  MoveL 3161 to (-403.79, 333.05, -22.06) mm, rotated rx -180 ry 0 rz 0.01 deg; joints [35.385, -31.602, 74.952, -134.407, 54.177, 150.081]
  MoveL 3162 to (-401.25, 328.08, -22.26) mm, rotated rx -180 ry 0 rz 0.01 deg; joints [35.301, -31.893, 75.575, -134.666, 54.367, 150.425]
  MoveL 3163 to (-395.74, 327.2, -22.47) mm, rotated rx -180 ry 0 rz 0.01 deg; joints [35.382, -32.188, 76.201, -134.749, 54.641, 150.663]
  MoveL 3164 to (-391.79, 331.15, -22.67) mm, rotated rx -180 ry 0 rz 0.01 deg; joints [35.561, -32.238, 76.316, -134.592, 54.778, 150.609]
  MoveL 3165 to (-392.66, 336.66, -22.87) mm, rotated rx 180 ry 0 rz 0.01 deg; joints [35.69, -31.995, 75.825, -134.331, 54.671, 150.312]
  MoveL 3166 to (-397.64, 339.2, -23.07) mm, rotated rx -180 ry 0 rz 0.01 deg; joints [35.663, -31.651, 75.129, -134.181, 54.411, 150.02]
  MoveL 3167 to (-398.51, 339.2, -23.1) mm, rotated rx -180 ry 0 rz 0.01 deg; joints [35.647, -31.606, 75.04, -134.175, 54.372, 149.991]
  MoveL 3168 to (-399.34, 339.13, -23.13) mm, rotated rx 180 ry 0 rz 0.01 deg; joints [35.629, -31.566, 74.959, -134.172, 54.334, 149.966]
  MoveL 3169 to (-399.69, 339.08, -23.14) mm, rotated rx 180 ry 0 rz 0.01 deg; joints [35.621, -31.55, 74.927, -134.173, 54.319, 149.957]
  MoveL 3170 to (-400.55, 338.85, -23.18) mm, rotated rx 180 ry 0 rz 0.01 deg; joints [35.599, -31.513, 74.855, -134.177, 54.282, 149.939]
  MoveL 3171 to (-400.6, 338.83, -23.18) mm, rotated rx 180 ry 0 rz 0.01 deg; joints [35.598, -31.512, 74.851, -134.178, 54.281, 149.938]
  MoveL 3172 to (-401.28, 338.49, -23.2) mm, rotated rx -180 ry 0 rz 0.01 deg; joints [35.576, -31.488, 74.805, -134.189, 54.254, 149.932]
  MoveL 3173 to (-401.4, 338.42, -23.21) mm, rotated rx -180 ry 0 rz 0.01 deg; joints [35.572, -31.484, 74.798, -134.192, 54.249, 149.932]
  MoveL 3174 to (-402.84, 337.05, -23.28) mm, rotated rx -180 ry 0 rz 0.01 deg; joints [35.509, -31.457, 74.75, -134.247, 54.202, 149.953]
  MoveL 3175 to (-402.87, 337.02, -23.28) mm, rotated rx 180 ry 0 rz 0.01 deg; joints [35.507, -31.457, 74.75, -134.249, 54.201, 149.954]
  MoveL 3176 to (-403.75, 334.43, -23.38) mm, rotated rx 180 ry 0 rz 0.01 deg; joints [35.422, -31.499, 74.848, -134.367, 54.196, 150.056]
  MoveL 3177 to (-403.78, 333.95, -23.39) mm, rotated rx 180 ry 0 rz 0.01 deg; joints [35.409, -31.514, 74.881, -134.39, 54.202, 150.08]
  MoveL 3178 to (-403.79, 333.65, -23.4) mm, rotated rx 180 ry 0 rz 0.01 deg; joints [35.401, -31.524, 74.902, -134.404, 54.206, 150.095]
  MoveL 3179 to (-403.79, 333.05, -23.43) mm, rotated rx -180 ry 0 rz 0.01 deg; joints [35.385, -31.544, 74.946, -134.434, 54.214, 150.126]
  MoveL 3180 to (-401.25, 328.08, -23.63) mm, rotated rx -180 ry 0 rz 0.01 deg; joints [35.302, -31.835, 75.57, -134.692, 54.404, 150.471]
  MoveL 3181 to (-395.74, 327.2, -23.83) mm, rotated rx -180 ry 0 rz 0.01 deg; joints [35.382, -32.13, 76.196, -134.775, 54.678, 150.709]
  MoveL 3182 to (-391.79, 331.15, -24.03) mm, rotated rx -180 ry 0 rz 0.01 deg; joints [35.562, -32.18, 76.31, -134.618, 54.815, 150.654]
  MoveL 3183 to (-392.66, 336.66, -24.23) mm, rotated rx -180 ry 0 rz 0.01 deg; joints [35.691, -31.937, 75.82, -134.357, 54.708, 150.358]
  MoveL 3184 to (-397.64, 339.2, -24.44) mm, rotated rx -180 ry 0 rz 0.01 deg; joints [35.664, -31.593, 75.124, -134.207, 54.448, 150.066]
  MoveL 3185 to (-398.51, 339.2, -24.47) mm, rotated rx -180 ry 0 rz 0.01 deg; joints [35.647, -31.549, 75.034, -134.201, 54.408, 150.036]
  MoveL 3186 to (-399.34, 339.13, -24.5) mm, rotated rx 180 ry 0 rz 0.01 deg; joints [35.63, -31.508, 74.954, -134.198, 54.371, 150.012]
  MoveL 3187 to (-399.69, 339.08, -24.51) mm, rotated rx 180 ry 0 rz 0.01 deg; joints [35.622, -31.492, 74.921, -134.199, 54.356, 150.002]
  MoveL 3188 to (-400.55, 338.85, -24.54) mm, rotated rx 180 ry 0 rz 0.01 deg; joints [35.6, -31.455, 74.849, -134.204, 54.319, 149.985]
  MoveL 3189 to (-400.6, 338.83, -24.54) mm, rotated rx 180 ry 0 rz 0.01 deg; joints [35.598, -31.454, 74.846, -134.204, 54.317, 149.984]
  MoveL 3190 to (-401.28, 338.49, -24.57) mm, rotated rx -180 ry 0 rz 0.01 deg; joints [35.577, -31.43, 74.8, -134.216, 54.29, 149.978]
  MoveL 3191 to (-401.4, 338.42, -24.57) mm, rotated rx -180 ry 0 rz 0.01 deg; joints [35.572, -31.426, 74.793, -134.218, 54.286, 149.978]
  MoveL 3192 to (-402.84, 337.05, -24.64) mm, rotated rx 180 ry 0 rz 0.01 deg; joints [35.509, -31.399, 74.744, -134.274, 54.238, 149.998]
  MoveL 3193 to (-402.87, 337.02, -24.64) mm, rotated rx -180 ry 0 rz 0.01 deg; joints [35.508, -31.399, 74.744, -134.275, 54.238, 149.999]
  MoveL 3194 to (-403.75, 334.43, -24.74) mm, rotated rx -180 ry 0 rz 0.01 deg; joints [35.423, -31.441, 74.843, -134.393, 54.233, 150.102]
  MoveL 3195 to (-403.78, 333.95, -24.76) mm, rotated rx -180 ry 0 rz 0.01 deg; joints [35.41, -31.456, 74.876, -134.417, 54.239, 150.126]
  MoveL 3196 to (-403.79, 333.65, -24.77) mm, rotated rx -180 ry 0 rz 0.01 deg; joints [35.402, -31.466, 74.896, -134.431, 54.242, 150.141]
  MoveL 3197 to (-403.79, 333.05, -24.79) mm, rotated rx -180 ry 0 rz 0.01 deg; joints [35.386, -31.486, 74.941, -134.46, 54.251, 150.172]
  MoveL 3198 to (-401.25, 328.08, -24.99) mm, rotated rx -180 ry 0 rz 0.01 deg; joints [35.302, -31.777, 75.564, -134.718, 54.441, 150.516]
  MoveL 3199 to (-395.74, 327.2, -25.19) mm, rotated rx 180 ry 0 rz 0.01 deg; joints [35.383, -32.072, 76.19, -134.8, 54.715, 150.754]
  MoveL 3200 to (-391.79, 331.15, -25.4) mm, rotated rx 180 ry 0 rz 0.01 deg; joints [35.562, -32.122, 76.305, -134.644, 54.852, 150.7]
  MoveL 3201 to (-392.66, 336.66, -25.6) mm, rotated rx -180 ry 0 rz 0.01 deg; joints [35.692, -31.879, 75.814, -134.383, 54.745, 150.403]
  MoveL 3202 to (-397.64, 339.2, -25.8) mm, rotated rx -180 ry 0 rz 0.01 deg; joints [35.664, -31.535, 75.118, -134.233, 54.485, 150.111]
  MoveL 3203 to (-398.51, 339.2, -25.83) mm, rotated rx -180 ry 0 rz 0.01 deg; joints [35.648, -31.491, 75.029, -134.227, 54.445, 150.082]
  MoveL 3204 to (-399.34, 339.13, -25.86) mm, rotated rx -180 ry 0 rz 0.01 deg; joints [35.631, -31.45, 74.948, -134.225, 54.408, 150.057]
  MoveL 3205 to (-399.69, 339.08, -25.87) mm, rotated rx 180 ry 0 rz 0.01 deg; joints [35.622, -31.434, 74.915, -134.225, 54.392, 150.048]
  MoveL 3206 to (-400.55, 338.85, -25.9) mm, rotated rx -180 ry 0 rz 0.01 deg; joints [35.6, -31.398, 74.843, -134.23, 54.356, 150.03]
  MoveL 3207 to (-400.6, 338.83, -25.91) mm, rotated rx -180 ry 0 rz 0.01 deg; joints [35.599, -31.396, 74.84, -134.23, 54.354, 150.03]
  MoveL 3208 to (-401.28, 338.49, -25.93) mm, rotated rx 180 ry 0 rz 0.01 deg; joints [35.577, -31.372, 74.794, -134.242, 54.327, 150.023]
  MoveL 3209 to (-401.4, 338.42, -25.94) mm, rotated rx -180 ry 0 rz 0.01 deg; joints [35.573, -31.369, 74.787, -134.245, 54.322, 150.023]
  MoveL 3210 to (-402.84, 337.05, -26.01) mm, rotated rx 180 ry 0 rz 0.01 deg; joints [35.51, -31.341, 74.739, -134.3, 54.275, 150.044]
  MoveL 3211 to (-402.87, 337.02, -26.01) mm, rotated rx 180 ry 0 rz 0.01 deg; joints [35.508, -31.341, 74.739, -134.301, 54.274, 150.045]
  MoveL 3212 to (-403.75, 334.43, -26.11) mm, rotated rx -180 ry 0 rz 0.01 deg; joints [35.424, -31.384, 74.837, -134.42, 54.27, 150.147]
  MoveL 3213 to (-403.78, 333.95, -26.12) mm, rotated rx 180 ry 0 rz 0.01 deg; joints [35.41, -31.398, 74.87, -134.443, 54.275, 150.171]
  MoveL 3214 to (-403.79, 333.65, -26.13) mm, rotated rx -180 ry 0 rz 0.01 deg; joints [35.403, -31.408, 74.891, -134.457, 54.279, 150.186]
  MoveL 3215 to (-403.79, 333.05, -26.15) mm, rotated rx -180 ry 0 rz 0.01 deg; joints [35.387, -31.428, 74.935, -134.486, 54.288, 150.217]
  MoveL 3216 to (-401.25, 328.08, -26.36) mm, rotated rx 180 ry 0 rz 0.01 deg; joints [35.303, -31.719, 75.558, -134.744, 54.478, 150.561]
  MoveL 3217 to (-395.74, 327.2, -26.56) mm, rotated rx -180 ry 0 rz 0.01 deg; joints [35.383, -32.013, 76.184, -134.826, 54.753, 150.799]
  MoveL 3218 to (-391.79, 331.15, -26.76) mm, rotated rx 180 ry 0 rz 0.01 deg; joints [35.563, -32.063, 76.299, -134.67, 54.89, 150.745]
  MoveL 3219 to (-392.66, 336.66, -26.96) mm, rotated rx 180 ry 0 rz 0.01 deg; joints [35.692, -31.821, 75.808, -134.409, 54.782, 150.449]
  MoveL 3220 to (-397.64, 339.2, -27.17) mm, rotated rx -180 ry 0 rz 0.01 deg; joints [35.665, -31.477, 75.112, -134.259, 54.521, 150.157]
  MoveL 3221 to (-398.51, 339.2, -27.2) mm, rotated rx -180 ry 0 rz 0.01 deg; joints [35.648, -31.433, 75.023, -134.253, 54.482, 150.127]
  MoveL 3222 to (-399.34, 339.13, -27.23) mm, rotated rx -180 ry 0 rz 0.01 deg; joints [35.631, -31.392, 74.942, -134.251, 54.444, 150.103]
  MoveL 3223 to (-399.69, 339.08, -27.24) mm, rotated rx -180 ry 0 rz 0.01 deg; joints [35.623, -31.376, 74.909, -134.251, 54.429, 150.093]
  MoveL 3224 to (-400.55, 338.85, -27.27) mm, rotated rx -180 ry 0 rz 0.01 deg; joints [35.601, -31.34, 74.837, -134.256, 54.392, 150.076]
  MoveL 3225 to (-400.6, 338.83, -27.27) mm, rotated rx -180 ry 0 rz 0.01 deg; joints [35.599, -31.338, 74.834, -134.256, 54.391, 150.075]
  MoveL 3226 to (-401.28, 338.49, -27.3) mm, rotated rx -180 ry 0 rz 0.01 deg; joints [35.578, -31.314, 74.788, -134.268, 54.364, 150.069]
  MoveL 3227 to (-401.4, 338.42, -27.3) mm, rotated rx -180 ry 0 rz 0.01 deg; joints [35.573, -31.311, 74.781, -134.271, 54.359, 150.069]
  MoveL 3228 to (-402.84, 337.05, -27.37) mm, rotated rx 180 ry 0 rz 0.01 deg; joints [35.51, -31.284, 74.733, -134.326, 54.311, 150.089]
  MoveL 3229 to (-402.87, 337.02, -27.37) mm, rotated rx -180 ry 0 rz 0.01 deg; joints [35.509, -31.283, 74.733, -134.327, 54.311, 150.09]
  MoveL 3230 to (-403.75, 334.43, -27.47) mm, rotated rx 180 ry 0 rz 0.01 deg; joints [35.424, -31.326, 74.831, -134.446, 54.306, 150.193]
  MoveL 3231 to (-403.78, 333.95, -27.49) mm, rotated rx -180 ry 0 rz 0.01 deg; joints [35.411, -31.341, 74.864, -134.469, 54.312, 150.217]
  MoveL 3232 to (-403.79, 333.65, -27.5) mm, rotated rx -180 ry 0 rz 0.01 deg; joints [35.403, -31.35, 74.885, -134.483, 54.316, 150.232]
  MoveL 3233 to (-403.79, 333.05, -27.52) mm, rotated rx 180 ry 0 rz 0.01 deg; joints [35.387, -31.37, 74.929, -134.512, 54.324, 150.263]
  MoveL 3234 to (-401.25, 328.08, -27.72) mm, rotated rx -180 ry 0 rz 0.01 deg; joints [35.303, -31.661, 75.552, -134.77, 54.515, 150.606]
  MoveL 3235 to (-395.74, 327.2, -27.92) mm, rotated rx -180 ry 0 rz 0.01 deg; joints [35.384, -31.955, 76.178, -134.852, 54.79, 150.845]
  MoveL 3236 to (-391.79, 331.15, -28.13) mm, rotated rx -180 ry 0 rz 0.01 deg; joints [35.563, -32.005, 76.293, -134.695, 54.927, 150.79]
  MoveL 3237 to (-392.66, 336.66, -28.33) mm, rotated rx 180 ry 0 rz 0.01 deg; joints [35.693, -31.763, 75.802, -134.435, 54.818, 150.494]
  MoveL 3238 to (-397.64, 339.2, -28.53) mm, rotated rx -180 ry 0 rz 0.01 deg; joints [35.665, -31.419, 75.106, -134.285, 54.558, 150.202]
  MoveL 3239 to (-398.51, 339.2, -28.56) mm, rotated rx 180 ry 0 rz 0.01 deg; joints [35.649, -31.375, 75.017, -134.279, 54.518, 150.173]
  MoveL 3240 to (-399.34, 339.13, -28.59) mm, rotated rx -180 ry 0 rz 0.01 deg; joints [35.632, -31.334, 74.936, -134.277, 54.481, 150.148]
  MoveL 3241 to (-399.69, 339.08, -28.6) mm, rotated rx 180 ry 0 rz 0.01 deg; joints [35.623, -31.318, 74.903, -134.277, 54.465, 150.139]
  MoveL 3242 to (-400.55, 338.85, -28.63) mm, rotated rx 180 ry 0 rz 0.01 deg; joints [35.601, -31.282, 74.831, -134.282, 54.429, 150.121]
  MoveL 3243 to (-400.6, 338.83, -28.64) mm, rotated rx 180 ry 0 rz 0.01 deg; joints [35.6, -31.28, 74.828, -134.282, 54.427, 150.12]
  MoveL 3244 to (-401.28, 338.49, -28.66) mm, rotated rx -180 ry 0 rz 0.01 deg; joints [35.578, -31.256, 74.782, -134.294, 54.4, 150.114]
  MoveL 3245 to (-401.4, 338.42, -28.67) mm, rotated rx -180 ry 0 rz 0.01 deg; joints [35.574, -31.253, 74.775, -134.297, 54.395, 150.114]
  MoveL 3246 to (-402.84, 337.05, -28.74) mm, rotated rx 180 ry 0 rz 0.01 deg; joints [35.511, -31.226, 74.726, -134.352, 54.348, 150.134]
  MoveL 3247 to (-402.87, 337.02, -28.74) mm, rotated rx -180 ry 0 rz 0.01 deg; joints [35.51, -31.225, 74.726, -134.353, 54.347, 150.135]
  MoveL 3248 to (-403.75, 334.43, -28.84) mm, rotated rx 180 ry 0 rz 0.01 deg; joints [35.425, -31.268, 74.825, -134.472, 54.343, 150.238]
  MoveL 3249 to (-403.78, 333.95, -28.85) mm, rotated rx 180 ry 0 rz 0.01 deg; joints [35.412, -31.282, 74.858, -134.495, 54.349, 150.262]
  MoveL 3250 to (-403.79, 333.65, -28.86) mm, rotated rx 180 ry 0 rz 0.01 deg; joints [35.404, -31.292, 74.878, -134.509, 54.352, 150.277]
  MoveL 3251 to (-403.79, 333.05, -28.88) mm, rotated rx -180 ry 0 rz 0.01 deg; joints [35.388, -31.312, 74.923, -134.538, 54.361, 150.308]
  MoveL 3252 to (-401.25, 328.08, -29.09) mm, rotated rx 180 ry 0 rz 0.01 deg; joints [35.304, -31.603, 75.546, -134.796, 54.552, 150.651]
  MoveL 3253 to (-395.74, 327.2, -29.29) mm, rotated rx 180 ry 0 rz 0.01 deg; joints [35.385, -31.897, 76.172, -134.877, 54.827, 150.89]
  MoveL 3254 to (-391.79, 331.15, -29.49) mm, rotated rx -180 ry 0 rz 0.01 deg; joints [35.564, -31.946, 76.287, -134.721, 54.964, 150.835]
  MoveL 3255 to (-392.66, 336.66, -29.69) mm, rotated rx -180 ry 0 rz 0.01 deg; joints [35.693, -31.704, 75.796, -134.46, 54.855, 150.539]
  MoveL 3256 to (-397.64, 339.2, -29.9) mm, rotated rx -180 ry 0 rz 0.01 deg; joints [35.666, -31.361, 75.1, -134.311, 54.595, 150.247]
  MoveL 3257 to (-398.51, 339.2, -29.93) mm, rotated rx 180 ry 0 rz 0.01 deg; joints [35.65, -31.316, 75.01, -134.305, 54.555, 150.218]
  MoveL 3258 to (-399.34, 339.13, -29.95) mm, rotated rx -180 ry 0 rz 0.01 deg; joints [35.632, -31.276, 74.93, -134.302, 54.517, 150.193]
  MoveL 3259 to (-399.69, 339.08, -29.97) mm, rotated rx 180 ry 0 rz 0.01 deg; joints [35.624, -31.26, 74.897, -134.303, 54.502, 150.184]
  MoveL 3260 to (-400.55, 338.85, -30) mm, rotated rx 180 ry 0 rz 0.01 deg; joints [35.602, -31.224, 74.825, -134.308, 54.465, 150.166]
  MoveL 3261 to (-400.6, 338.83, -30) mm, rotated rx 180 ry 0 rz 0.01 deg; joints [35.601, -31.222, 74.822, -134.308, 54.464, 150.166]
  MoveL 3262 to (-400.13, 339.01, -30) mm, rotated rx -180 ry 0 rz 0.01 deg; joints [35.614, -31.239, 74.856, -134.303, 54.483, 150.173]
  MoveL 3263 to (-398.92, 339.2, -30) mm, rotated rx 180 ry 0 rz 0.01 deg; joints [35.642, -31.292, 74.967, -134.303, 54.537, 150.206]
  MoveL 3264 to (-213.26, 339.2, -30) mm, rotated rx -180 ry 0 rz 0.01 deg; joints [39.465, -39.376, 91.77, -134.189, 62.458, 155.431]
  MoveL 3265 to (-213.59, 339.15, -30) mm, rotated rx -180 ry 0 rz 0.01 deg; joints [39.457, -39.365, 91.748, -134.194, 62.446, 155.425]
  MoveL 3266 to (-214.12, 339.03, -30) mm, rotated rx -180 ry 0 rz 0.01 deg; joints [39.441, -39.349, 91.713, -134.203, 62.426, 155.418]
  MoveL 3267 to (-215.21, 338.67, -30) mm, rotated rx 180 ry 0 rz 0.01 deg; joints [39.407, -39.318, 91.649, -134.225, 62.388, 155.407]
  MoveL 3268 to (-215.66, 338.49, -30) mm, rotated rx 180 ry 0 rz 0.01 deg; joints [39.392, -39.306, 91.624, -134.235, 62.373, 155.404]
  MoveL 3269 to (-226.55, 333.14, -30) mm, rotated rx 180 ry 0 rz 0.01 deg; joints [39.004, -39.05, 91.096, -134.527, 62.012, 155.373]
  MoveL 3270 to (-227.09, 332.81, -30) mm, rotated rx -180 ry 0 rz 0.01 deg; joints [38.983, -39.039, 91.074, -134.545, 61.995, 155.374]
  MoveL 3271 to (-228.18, 331.99, -30) mm, rotated rx 180 ry 0 rz 0.01 deg; joints [38.936, -39.022, 91.039, -134.585, 61.962, 155.382]
  MoveL 3272 to (-228.47, 331.74, -30) mm, rotated rx 180 ry 0 rz 0.01 deg; joints [38.923, -39.018, 91.032, -134.597, 61.954, 155.386]
  MoveL 3273 to (-236.6, 324.01, -30) mm, rotated rx -180 ry 0 rz 0.01 deg; joints [38.532, -38.937, 90.874, -134.967, 61.729, 155.516]
  MoveL 3274 to (-236.83, 323.76, -30) mm, rotated rx 180 ry 0 rz 0.01 deg; joints [38.52, -38.936, 90.871, -134.978, 61.722, 155.521]
  MoveL 3275 to (-237.77, 322.67, -30) mm, rotated rx 180 ry 0 rz 0.01 deg; joints [38.47, -38.932, 90.865, -135.029, 61.699, 155.544]
  MoveL 3276 to (-238.12, 322.17, -30) mm, rotated rx -180 ry 0 rz 0.01 deg; joints [38.449, -38.934, 90.868, -135.052, 61.691, 155.556]
  MoveL 3277 to (-240.45, 318.18, -30) mm, rotated rx -180 ry 0 rz 0.01 deg; joints [38.288, -38.963, 90.937, -135.231, 61.649, 155.667]
  MoveL 3278 to (-240.5, 318.08, -30) mm, rotated rx -180 ry 0 rz 0.01 deg; joints [38.284, -38.964, 90.938, -135.235, 61.648, 155.67]
  MoveL 3279 to (-244.03, 311.56, -30) mm, rotated rx -180 ry 0 rz 0.01 deg; joints [38.027, -39.023, 91.07, -135.526, 61.589, 155.856]
  MoveL 3280 to (-244.21, 311.15, -30) mm, rotated rx -180 ry 0 rz 0.01 deg; joints [38.012, -39.027, 91.081, -135.544, 61.586, 155.868]
  MoveL 3281 to (-244.76, 309.7, -30) mm, rotated rx 180 ry 0 rz 0.01 deg; joints [37.96, -39.049, 91.129, -135.607, 61.582, 155.915]
  MoveL 3282 to (-244.95, 309.01, -30) mm, rotated rx 180 ry 0 rz 0.01 deg; joints [37.936, -39.063, 91.158, -135.637, 61.584, 155.939]
  MoveL 3283 to (-246.39, 299.58, -30) mm, rotated rx -180 ry 0 rz 0.01 deg; joints [37.643, -39.287, 91.642, -136.037, 61.644, 156.292]
  MoveL 3284 to (-246.42, 299.36, -30) mm, rotated rx -180 ry 0 rz 0.01 deg; joints [37.636, -39.293, 91.654, -136.046, 61.646, 156.3]
  MoveL 3285 to (-246.51, 298.27, -30) mm, rotated rx 180 ry 0 rz 0.01 deg; joints [37.603, -39.321, 91.715, -136.092, 61.656, 156.342]
  MoveC 3286 to (-246.51, 297.75, -30) mm, rotated rx -180 ry 0 rz 0.01 deg; joints [37.589, -39.336, 91.748, -136.113, 61.662, 156.363] to (-246.44, 297.24, -30) mm, rotated rx 180 ry 0 rz 0.01 deg; joints [37.576, -39.354, 91.786, -136.134, 61.672, 156.385]
  MoveL 3287 to (-245.04, 290.99, -30) mm, rotated rx 180 ry 0 rz 0.01 deg; joints [37.431, -39.593, 92.296, -136.384, 61.806, 156.671]
  MoveL 3288 to (-245.03, 290.92, -30) mm, rotated rx -180 ry 0 rz 0.01 deg; joints [37.429, -39.596, 92.301, -136.387, 61.808, 156.674]
  MoveL 3289 to (-244.07, 287.01, -30) mm, rotated rx 180 ry 0 rz 0.01 deg; joints [37.34, -39.747, 92.625, -136.543, 61.895, 156.852]
  MoveL 3290 to (-243.75, 286.2, -30) mm, rotated rx 180 ry 0 rz 0.01 deg; joints [37.324, -39.783, 92.702, -136.574, 61.918, 156.892]
  MoveL 3291 to (-241.96, 282.93, -30) mm, rotated rx -180 ry 0 rz 0.01 deg; joints [37.27, -39.948, 93.051, -136.698, 62.031, 157.063]
  MoveL 3292 to (-241.77, 282.61, -30) mm, rotated rx -180 ry 0 rz 0.01 deg; joints [37.265, -39.965, 93.088, -136.71, 62.043, 157.08]
  MoveL 3293 to (-239.73, 279.71, -30) mm, rotated rx -180 ry 0 rz 0.01 deg; joints [37.227, -40.128, 93.434, -136.816, 62.16, 157.241]
  MoveL 3294 to (-239.54, 279.46, -30) mm, rotated rx -180 ry 0 rz 0.01 deg; joints [37.224, -40.142, 93.464, -136.824, 62.171, 157.255]
  MoveL 3295 to (-237.07, 276.56, -30) mm, rotated rx -180 ry 0 rz 0.01 deg; joints [37.194, -40.321, 93.844, -136.927, 62.306, 157.425]
  MoveL 3296 to (-236.53, 276.05, -30) mm, rotated rx -180 ry 0 rz 0.01 deg; joints [37.192, -40.356, 93.919, -136.944, 62.333, 157.457]
  MoveL 3297 to (-232.69, 273.15, -30) mm, rotated rx -180 ry 0 rz 0.01 deg; joints [37.192, -40.587, 94.408, -137.036, 62.523, 157.655]
  MoveL 3298 to (-232.49, 273.01, -30) mm, rotated rx 180 ry 0 rz 0.01 deg; joints [37.192, -40.599, 94.433, -137.04, 62.532, 157.665]
  MoveL 3299 to (-229.8, 271.26, -30) mm, rotated rx 180 ry 0 rz 0.01 deg; joints [37.201, -40.752, 94.757, -137.092, 62.661, 157.792]
  MoveL 3300 to (-229.47, 271.08, -30) mm, rotated rx 180 ry 0 rz 0.01 deg; joints [37.203, -40.769, 94.794, -137.097, 62.676, 157.806]
  MoveL 3301 to (-227.17, 269.92, -30) mm, rotated rx -180 ry 0 rz 0.01 deg; joints [37.22, -40.89, 95.049, -137.126, 62.782, 157.901]
  MoveL 3302 to (-226.75, 269.75, -30) mm, rotated rx -180 ry 0 rz 0.01 deg; joints [37.224, -40.911, 95.093, -137.13, 62.8, 157.917]
  MoveL 3303 to (-223.98, 268.79, -30) mm, rotated rx 180 ry 0 rz 0.01 deg; joints [37.257, -41.043, 95.374, -137.148, 62.921, 158.014]
  MoveL 3304 to (-223.48, 268.66, -30) mm, rotated rx -180 ry 0 rz 0.01 deg; joints [37.264, -41.066, 95.421, -137.149, 62.943, 158.03]
  MoveL 3305 to (-219.13, 267.87, -30) mm, rotated rx 180 ry 0 rz 0.01 deg; joints [37.337, -41.253, 95.816, -137.146, 63.124, 158.154]
  MoveL 3306 to (-218.95, 267.85, -30) mm, rotated rx 180 ry 0 rz 0.01 deg; joints [37.34, -41.261, 95.832, -137.146, 63.131, 158.159]
  MoveL 3307 to (-215.32, 267.39, -30) mm, rotated rx 180 ry 0 rz 0.01 deg; joints [37.406, -41.41, 96.148, -137.134, 63.279, 158.253]
  MoveL 3308 to (-214.9, 267.36, -30) mm, rotated rx 180 ry 0 rz 0.01 deg; joints [37.415, -41.427, 96.183, -137.131, 63.296, 158.263]
  MoveL 3309 to (-178.62, 267.36, -30) mm, rotated rx -180 ry 0 rz 0.01 deg; joints [38.23, -42.764, 99.002, -136.789, 64.694, 159.014]
  MoveL 3310 to (-178.19, 267.39, -30) mm, rotated rx 180 ry 0 rz 0.01 deg; joints [38.24, -42.778, 99.033, -136.784, 64.71, 159.021]
  MoveL 3311 to (-174.57, 267.85, -30) mm, rotated rx -180 ry 0 rz 0.01 deg; joints [38.336, -42.896, 99.282, -136.727, 64.842, 159.077]
  MoveL 3312 to (-174.39, 267.87, -30) mm, rotated rx 180 ry 0 rz 0.01 deg; joints [38.341, -42.902, 99.294, -136.724, 64.849, 159.08]
  MoveL 3313 to (-170.03, 268.66, -30) mm, rotated rx -180 ry 0 rz 0.01 deg; joints [38.465, -43.036, 99.577, -136.646, 65.003, 159.138]
  MoveL 3314 to (-169.59, 268.78, -30) mm, rotated rx 180 ry 0 rz 0.01 deg; joints [38.478, -43.049, 99.604, -136.637, 65.019, 159.142]
  MoveL 3315 to (-167.47, 269.46, -30) mm, rotated rx -180 ry 0 rz 0.01 deg; joints [38.547, -43.106, 99.722, -136.586, 65.09, 159.159]
  MoveL 3316 to (-167.12, 269.6, -30) mm, rotated rx 180 ry 0 rz 0.01 deg; joints [38.559, -43.115, 99.74, -136.577, 65.101, 159.161]
  MoveL 3317 to (-164.88, 270.63, -30) mm, rotated rx 180 ry 0 rz 0.01 deg; joints [38.641, -43.166, 99.848, -136.511, 65.173, 159.167]
  MoveL 3318 to (-164.5, 270.83, -30) mm, rotated rx -180 ry 0 rz 0.01 deg; joints [38.656, -43.174, 99.864, -136.499, 65.184, 159.167]
  MoveL 3319 to (-161.59, 272.64, -30) mm, rotated rx 180 ry 0 rz 0.01 deg; joints [38.776, -43.227, 99.974, -136.395, 65.271, 159.158]
  MoveL 3320 to (-161.36, 272.79, -30) mm, rotated rx 180 ry 0 rz 0.01 deg; joints [38.786, -43.231, 99.982, -136.386, 65.277, 159.156]
  MoveL 3321 to (-157, 276.04, -30) mm, rotated rx 180 ry 0 rz 0.01 deg; joints [38.981, -43.295, 100.113, -136.208, 65.4, 159.122]
  MoveL 3322 to (-156.45, 276.55, -30) mm, rotated rx 180 ry 0 rz 0.01 deg; joints [39.009, -43.301, 100.123, -136.181, 65.414, 159.113]
  MoveL 3323 to (-154.49, 278.84, -30) mm, rotated rx 180 ry 0 rz 0.01 deg; joints [39.121, -43.306, 100.131, -136.067, 65.458, 159.066]
  MoveL 3324 to (-154.32, 279.05, -30) mm, rotated rx 180 ry 0 rz 0.01 deg; joints [39.131, -43.306, 100.13, -136.057, 65.462, 159.062]
  MoveL 3325 to (-151.94, 282.32, -30) mm, rotated rx -180 ry 0 rz 0.01 deg; joints [39.282, -43.298, 100.109, -135.9, 65.509, 158.987]
  MoveL 3326 to (-151.71, 282.67, -30) mm, rotated rx 180 ry 0 rz 0.01 deg; joints [39.297, -43.296, 100.105, -135.884, 65.513, 158.978]
  MoveL 3327 to (-149.77, 286.18, -30) mm, rotated rx 180 ry 0 rz 0.01 deg; joints [39.444, -43.266, 100.035, -135.722, 65.541, 158.885]
  MoveL 3328 to (-149.44, 287.04, -30) mm, rotated rx -180 ry 0 rz 0.01 deg; joints [39.477, -43.254, 100.008, -135.684, 65.543, 158.859]
  MoveL 3329 to (-147.12, 296.83, -30) mm, rotated rx 180 ry 0 rz 0.01 deg; joints [39.812, -43.058, 99.578, -135.27, 65.505, 158.534]
  MoveL 3330 to (-147.03, 297.45, -30) mm, rotated rx -180 ry 0 rz 0.01 deg; joints [39.831, -43.043, 99.546, -135.244, 65.501, 158.513]
  MoveL 3331 to (-146.99, 298.18, -30) mm, rotated rx 180 ry 0 rz 0.01 deg; joints [39.853, -43.024, 99.504, -135.215, 65.493, 158.486]
  MoveL 3332 to (-147.03, 298.84, -30) mm, rotated rx 180 ry 0 rz 0.01 deg; joints [39.871, -43.004, 99.46, -135.19, 65.483, 158.46]
  MoveL 3333 to (-148.48, 308.63, -30) mm, rotated rx -180 ry 0 rz 0.01 deg; joints [40.114, -42.671, 98.742, -134.819, 65.306, 158.055]
  MoveL 3334 to (-148.63, 309.25, -30) mm, rotated rx -180 ry 0 rz 0.01 deg; joints [40.128, -42.647, 98.692, -134.796, 65.293, 158.028]
  MoveL 3335 to (-149.27, 311.07, -30) mm, rotated rx -180 ry 0 rz 0.01 deg; joints [40.164, -42.572, 98.53, -134.732, 65.246, 157.945]
  MoveL 3336 to (-149.48, 311.55, -30) mm, rotated rx -180 ry 0 rz 0.01 deg; joints [40.172, -42.551, 98.484, -134.715, 65.232, 157.922]
  MoveL 3337 to (-151.43, 315.17, -30) mm, rotated rx 180 ry 0 rz 0.01 deg; joints [40.228, -42.376, 98.11, -134.593, 65.115, 157.742]
  MoveL 3338 to (-151.46, 315.23, -30) mm, rotated rx -180 ry 0 rz 0.01 deg; joints [40.229, -42.373, 98.105, -134.591, 65.113, 157.739]
  MoveL 3339 to (-155.12, 321.76, -30) mm, rotated rx 180 ry 0 rz 0.01 deg; joints [40.325, -42.051, 97.416, -134.373, 64.894, 157.408]
  MoveL 3340 to (-155.44, 322.24, -30) mm, rotated rx 180 ry 0 rz 0.01 deg; joints [40.33, -42.026, 97.361, -134.357, 64.876, 157.383]
  MoveL 3341 to (-156.62, 323.69, -30) mm, rotated rx -180 ry 0 rz 0.01 deg; joints [40.343, -41.941, 97.18, -134.312, 64.814, 157.301]
  MoveL 3342 to (-156.92, 324.01, -30) mm, rotated rx -180 ry 0 rz 0.01 deg; joints [40.345, -41.921, 97.138, -134.303, 64.799, 157.283]
  MoveL 3343 to (-165.04, 331.74, -30) mm, rotated rx -180 ry 0 rz 0.01 deg; joints [40.368, -41.398, 96.026, -134.079, 64.398, 156.805]
  MoveL 3344 to (-165.34, 331.99, -30) mm, rotated rx -180 ry 0 rz 0.01 deg; joints [40.368, -41.38, 95.987, -134.072, 64.384, 156.789]
  MoveL 3345 to (-166.42, 332.81, -30) mm, rotated rx 180 ry 0 rz 0.01 deg; joints [40.365, -41.316, 95.851, -134.05, 64.333, 156.733]
  MoveL 3346 to (-166.97, 333.14, -30) mm, rotated rx -180 ry 0 rz 0.01 deg; joints [40.361, -41.286, 95.789, -134.042, 64.308, 156.708]
  MoveL 3347 to (-177.85, 338.49, -30) mm, rotated rx -180 ry 0 rz 0.01 deg; joints [40.254, -40.727, 94.606, -133.931, 63.83, 156.257]
  MoveL 3348 to (-178.19, 338.64, -30) mm, rotated rx 180 ry 0 rz 0.01 deg; joints [40.251, -40.711, 94.57, -133.929, 63.815, 156.244]
  MoveL 3349 to (-178.91, 338.9, -30) mm, rotated rx -180 ry 0 rz 0.01 deg; joints [40.241, -40.676, 94.497, -133.925, 63.784, 156.217]
  MoveL 3350 to (-179.55, 339.06, -30) mm, rotated rx 180 ry 0 rz 0.01 deg; joints [40.231, -40.648, 94.437, -133.924, 63.758, 156.196]
  MoveL 3351 to (-180.46, 339.2, -30) mm, rotated rx 180 ry 0 rz 0.01 deg; joints [40.213, -40.61, 94.357, -133.927, 63.722, 156.171]
  MoveL 3352 to (4.87, 339.21, -30) mm, rotated rx -180 ry 0 rz 0.01 deg; joints [44.913, -46.774, 107.418, -131.39, 70.267, 159.8]
  MoveL 3353 to (5.94, 339.15, -30) mm, rotated rx 180 ry 0 rz 0.01 deg; joints [44.941, -46.808, 107.491, -131.373, 70.303, 159.821]
  MoveL 3354 to (6.8, 338.95, -30) mm, rotated rx 180 ry 0 rz 0.01 deg; joints [44.959, -46.84, 107.559, -131.364, 70.333, 159.843]
  MoveL 3355 to (7.07, 338.84, -30) mm, rotated rx -180 ry 0 rz 0.01 deg; joints [44.963, -46.851, 107.583, -131.363, 70.344, 159.852]
  MoveL 3356 to (7.37, 338.63, -30) mm, rotated rx -180 ry 0 rz 0.01 deg; joints [44.966, -46.866, 107.616, -131.365, 70.356, 159.865]
  MoveL 3357 to (9.66, 336.38, -30) mm, rotated rx 180 ry 0 rz 0.01 deg; joints [44.967, -47, 107.906, -131.406, 70.46, 159.99]
  MoveL 3358 to (9.9, 336.02, -30) mm, rotated rx 180 ry 0 rz 0.01 deg; joints [44.963, -47.018, 107.944, -131.415, 70.472, 160.007]
  MoveL 3359 to (10.07, 335.56, -30) mm, rotated rx 180 ry 0 rz 0.01 deg; joints [44.955, -47.036, 107.984, -131.429, 70.484, 160.027]
  MoveL 3360 to (10.27, 334.35, -30) mm, rotated rx 180 ry 0 rz 0.01 deg; joints [44.927, -47.077, 108.074, -131.47, 70.506, 160.075]
  MoveL 3361 to (10.27, 31.84, -30) mm, rotated rx -180 ry 0 rz 0.01 deg; joints [35.126, -54.404, 124.671, -143.341, 74.579, 169.75]
  MoveL 3362 to (9.14, 36.48, -30) mm, rotated rx 180 ry 0 rz 0.01 deg; joints [35.269, -54.28, 124.38, -143.169, 74.475, 169.606]
  MoveL 3363 to (9.02, 36.86, -30) mm, rotated rx -180 ry 0 rz 0.01 deg; joints [35.28, -54.268, 124.354, -143.155, 74.466, 169.594]
  MoveL 3364 to (8.51, 38.24, -30) mm, rotated rx -180 ry 0 rz 0.01 deg; joints [35.317, -54.226, 124.256, -143.107, 74.428, 169.549]
  MoveL 3365 to (8.27, 38.74, -30) mm, rotated rx 180 ry 0 rz 0.01 deg; joints [35.33, -54.209, 124.217, -143.091, 74.413, 169.531]
  MoveL 3366 to (6.11, 42.48, -30) mm, rotated rx 180 ry 0 rz 0.01 deg; joints [35.411, -54.071, 123.899, -142.978, 74.286, 169.396]
  MoveL 3367 to (6.06, 42.56, -30) mm, rotated rx -180 ry 0 rz 0.01 deg; joints [35.413, -54.068, 123.892, -142.976, 74.283, 169.393]
  MoveL 3368 to (2.27, 48.73, -30) mm, rotated rx -180 ry 0 rz 0.01 deg; joints [35.54, -53.832, 123.35, -142.794, 74.066, 169.164]
  MoveL 3369 to (2.07, 49.02, -30) mm, rotated rx -180 ry 0 rz 0.01 deg; joints [35.545, -53.82, 123.323, -142.786, 74.055, 169.153]
  MoveL 3370 to (1.04, 50.35, -30) mm, rotated rx 180 ry 0 rz 0.01 deg; joints [35.567, -53.763, 123.192, -142.751, 74.001, 169.1]
  MoveL 3371 to (0.49, 50.92, -30) mm, rotated rx 180 ry 0 rz 0.01 deg; joints [35.573, -53.735, 123.128, -142.738, 73.974, 169.076]
  MoveL 3372 to (-7.44, 57.29, -30) mm, rotated rx -180 ry 0 rz 0.01 deg; joints [35.599, -53.37, 122.299, -142.631, 73.61, 168.775]
  MoveL 3373 to (-7.81, 57.56, -30) mm, rotated rx 180 ry 0 rz 0.01 deg; joints [35.599, -53.353, 122.261, -142.627, 73.593, 168.762]
  MoveL 3374 to (-8.48, 57.96, -30) mm, rotated rx -180 ry 0 rz 0.01 deg; joints [35.596, -53.325, 122.198, -142.624, 73.565, 168.74]
  MoveL 3375 to (-9.25, 58.3, -30) mm, rotated rx 180 ry 0 rz 0.01 deg; joints [35.589, -53.295, 122.13, -142.625, 73.533, 168.719]
  MoveL 3376 to (-19.1, 61.27, -30) mm, rotated rx -180 ry 0 rz 0.01 deg; joints [35.442, -52.937, 121.329, -142.693, 73.148, 168.482]
  MoveL 3377 to (-20, 61.42, -30) mm, rotated rx 180 ry 0 rz 0.01 deg; joints [35.425, -52.907, 121.262, -142.704, 73.115, 168.464]
  MoveL 3378 to (-23.26, 61.5, -30) mm, rotated rx 180 ry 0 rz 0.01 deg; joints [35.344, -52.807, 121.038, -142.763, 72.999, 168.411]
  MoveL 3379 to (-23.6, 61.49, -30) mm, rotated rx 180 ry 0 rz 0.01 deg; joints [35.335, -52.797, 121.016, -142.77, 72.987, 168.406]
  MoveL 3380 to (-27.23, 61.21, -30) mm, rotated rx 180 ry 0 rz 0.01 deg; joints [35.233, -52.692, 120.784, -142.851, 72.863, 168.358]
  MoveL 3381 to (-27.55, 61.17, -30) mm, rotated rx 180 ry 0 rz 0.01 deg; joints [35.224, -52.683, 120.765, -142.859, 72.853, 168.354]
  MoveL 3382 to (-31.54, 60.47, -30) mm, rotated rx 180 ry 0 rz 0.01 deg; joints [35.098, -52.575, 120.528, -142.962, 72.721, 168.312]
  MoveL 3383 to (-32.27, 60.26, -30) mm, rotated rx -180 ry 0 rz 0.01 deg; joints [35.072, -52.557, 120.488, -142.985, 72.698, 168.306]
  MoveL 3384 to (-36.67, 58.42, -30) mm, rotated rx 180 ry 0 rz 0.01 deg; joints [34.896, -52.46, 120.277, -143.143, 72.567, 168.29]
  MoveL 3385 to (-36.89, 58.31, -30) mm, rotated rx 180 ry 0 rz 0.01 deg; joints [34.886, -52.455, 120.267, -143.152, 72.561, 168.29]
  MoveL 3386 to (-40.11, 56.68, -30) mm, rotated rx 180 ry 0 rz 0.01 deg; joints [34.748, -52.389, 120.125, -143.279, 72.468, 168.286]
  MoveL 3387 to (-40.47, 56.47, -30) mm, rotated rx -180 ry 0 rz 0.01 deg; joints [34.731, -52.383, 120.11, -143.295, 72.458, 168.286]
  MoveL 3388 to (-42.35, 55.2, -30) mm, rotated rx -180 ry 0 rz 0.01 deg; joints [34.639, -52.35, 120.042, -143.382, 72.408, 168.293]
  MoveL 3389 to (-42.66, 54.97, -30) mm, rotated rx 180 ry 0 rz 0.01 deg; joints [34.623, -52.346, 120.032, -143.397, 72.4, 168.295]
  MoveL 3390 to (-44.72, 53.2, -30) mm, rotated rx 180 ry 0 rz 0.01 deg; joints [34.509, -52.318, 119.974, -143.508, 72.351, 168.313]
  MoveL 3391 to (-45.04, 52.88, -30) mm, rotated rx 180 ry 0 rz 0.01 deg; joints [34.489, -52.314, 119.967, -143.527, 72.343, 168.317]
  MoveL 3392 to (-46.91, 50.78, -30) mm, rotated rx -180 ry 0 rz 0.01 deg; joints [34.368, -52.299, 119.937, -143.649, 72.304, 168.347]
  MoveL 3393 to (-47.05, 50.61, -30) mm, rotated rx -180 ry 0 rz 0.01 deg; joints [34.358, -52.298, 119.935, -143.659, 72.302, 168.349]
  MoveL 3394 to (-50.38, 46.34, -30) mm, rotated rx 180 ry 0 rz 0.01 deg; joints [34.123, -52.28, 119.906, -143.897, 72.239, 168.418]
  MoveL 3395 to (-50.64, 45.95, -30) mm, rotated rx -180 ry 0 rz 0.01 deg; joints [34.103, -52.28, 119.906, -143.918, 72.235, 168.425]
  MoveL 3396 to (-68.79, 14.55, -30) mm, rotated rx 180 ry 0 rz 0.01 deg; joints [32.525, -52.325, 120.077, -145.558, 71.991, 169.014]
  MoveL 3397 to (-68.98, 14.18, -30) mm, rotated rx 180 ry 0 rz 0.01 deg; joints [32.507, -52.327, 120.08, -145.577, 71.989, 169.022]
  MoveL 3398 to (-70.67, 10.19, -30) mm, rotated rx -180 ry 0 rz 0.01 deg; joints [32.321, -52.349, 120.139, -145.775, 71.98, 169.104]
  MoveL 3399 to (-70.75, 9.99, -30) mm, rotated rx -180 ry 0 rz 0.01 deg; joints [32.312, -52.35, 120.142, -145.785, 71.979, 169.109]
  MoveL 3400 to (-72.02, 6.36, -30) mm, rotated rx 180 ry 0 rz 0.01 deg; joints [32.148, -52.379, 120.213, -145.961, 71.98, 169.187]
  MoveL 3401 to (-72.14, 5.94, -30) mm, rotated rx -180 ry 0 rz 0.01 deg; joints [32.13, -52.383, 120.223, -145.981, 71.981, 169.197]
  MoveL 3402 to (-72.6, 3.77, -30) mm, rotated rx 180 ry 0 rz 0.01 deg; joints [32.039, -52.409, 120.286, -146.081, 71.992, 169.249]
  MoveL 3403 to (-72.66, 3.38, -30) mm, rotated rx 180 ry 0 rz 0.01 deg; joints [32.023, -52.415, 120.299, -146.099, 71.995, 169.258]
  MoveL 3404 to (-72.93, 0.48, -30) mm, rotated rx -180 ry 0 rz 0.01 deg; joints [31.909, -52.46, 120.408, -146.227, 72.023, 169.332]
  MoveL 3405 to (-72.94, 0.01, -30) mm, rotated rx 180 ry 0 rz 0.01 deg; joints [31.891, -52.469, 120.427, -146.247, 72.029, 169.345]
  MoveL 3406 to (-72.81, -2.9, -30) mm, rotated rx -180 ry 0 rz 0.01 deg; joints [31.787, -52.527, 120.563, -146.369, 72.072, 169.424]
  MoveL 3407 to (-72.79, -3.12, -30) mm, rotated rx -180 ry 0 rz 0.01 deg; joints [31.779, -52.532, 120.574, -146.378, 72.075, 169.43]
  MoveL 3408 to (-72.17, -8.56, -30) mm, rotated rx 180 ry 0 rz 0.01 deg; joints [31.59, -52.652, 120.854, -146.601, 72.169, 169.584]
  MoveL 3409 to (-72, -9.3, -30) mm, rotated rx 180 ry 0 rz 0.01 deg; joints [31.566, -52.671, 120.898, -146.63, 72.185, 169.607]
  MoveL 3410 to (-70.79, -12.74, -30) mm, rotated rx 180 ry 0 rz 0.01 deg; joints [31.465, -52.773, 121.131, -146.757, 72.275, 169.715]
  MoveL 3411 to (-70.68, -13.03, -30) mm, rotated rx -180 ry 0 rz 0.01 deg; joints [31.457, -52.782, 121.152, -146.767, 72.283, 169.725]
  MoveL 3412 to (-69.26, -16.12, -30) mm, rotated rx 180 ry 0 rz 0.01 deg; joints [31.373, -52.883, 121.384, -146.876, 72.376, 169.827]
  MoveL 3413 to (-69.12, -16.4, -30) mm, rotated rx 180 ry 0 rz 0.01 deg; joints [31.366, -52.893, 121.406, -146.886, 72.385, 169.836]
  MoveL 3414 to (-67.66, -18.94, -30) mm, rotated rx 180 ry 0 rz 0.01 deg; joints [31.304, -52.985, 121.617, -146.97, 72.472, 169.924]
  MoveL 3415 to (-67.52, -19.15, -30) mm, rotated rx 180 ry 0 rz 0.01 deg; joints [31.299, -52.993, 121.636, -146.977, 72.48, 169.932]
  MoveL 3416 to (-66.77, -20.26, -30) mm, rotated rx -180 ry 0 rz 0.01 deg; joints [31.274, -53.037, 121.736, -147.012, 72.522, 169.972]
  MoveL 3417 to (-66.29, -20.83, -30) mm, rotated rx -180 ry 0 rz 0.01 deg; joints [31.264, -53.062, 121.794, -147.028, 72.547, 169.994]
  MoveL 3418 to (-59.76, -26.97, -30) mm, rotated rx 180 ry 0 rz 0.01 deg; joints [31.18, -53.378, 122.512, -147.182, 72.869, 170.249]
  MoveL 3419 to (-59.61, -27.11, -30) mm, rotated rx 180 ry 0 rz 0.01 deg; joints [31.179, -53.385, 122.529, -147.185, 72.877, 170.255]
  MoveL 3420 to (-58.52, -28.02, -30) mm, rotated rx 180 ry 0 rz 0.01 deg; joints [31.169, -53.436, 122.644, -147.206, 72.929, 170.295]
  MoveC 3421 to (-58.08, -28.32, -30) mm, rotated rx 180 ry 0 rz 0.01 deg; joints [31.168, -53.455, 122.687, -147.211, 72.949, 170.309] to (-57.61, -28.56, -30) mm, rotated rx -180 ry 0 rz 0.01 deg; joints [31.17, -53.474, 122.73, -147.213, 72.97, 170.322]
  MoveL 3422 to (-50.81, -31.27, -30) mm, rotated rx 180 ry 0 rz 0.01 deg; joints [31.224, -53.734, 123.319, -147.212, 73.256, 170.491]
  MoveL 3423 to (-342.73, -31.27, -30) mm, rotated rx -180 ry 0 rz 0.01 deg; joints [25.555, -43.349, 100.769, -150.599, 61.537, 166.051]
  MoveL 3424 to (-336.29, -28.75, -30) mm, rotated rx 180 ry 0 rz 0.01 deg; joints [25.744, -43.563, 101.219, -150.454, 61.792, 166.082]
  MoveL 3425 to (-335.78, -28.51, -30) mm, rotated rx 180 ry 0 rz 0.01 deg; joints [25.761, -43.579, 101.253, -150.44, 61.812, 166.083]
  MoveL 3426 to (-335.06, -28.07, -30) mm, rotated rx 180 ry 0 rz 0.01 deg; joints [25.787, -43.6, 101.297, -150.417, 61.839, 166.082]
  MoveL 3427 to (-334.48, -27.64, -30) mm, rotated rx 180 ry 0 rz 0.01 deg; joints [25.811, -43.615, 101.328, -150.395, 61.859, 166.079]
  MoveL 3428 to (-327.59, -21.19, -30) mm, rotated rx 180 ry 0 rz 0.01 deg; joints [26.142, -43.772, 101.649, -150.077, 62.089, 165.997]
  MoveL 3429 to (-327.4, -20.99, -30) mm, rotated rx 180 ry 0 rz 0.01 deg; joints [26.152, -43.776, 101.657, -150.067, 62.095, 165.995]
  MoveL 3430 to (-326.75, -20.28, -30) mm, rotated rx -180 ry 0 rz 0.01 deg; joints [26.187, -43.789, 101.683, -150.032, 62.116, 165.984]
  MoveL 3431 to (-326.35, -19.74, -30) mm, rotated rx 180 ry 0 rz 0.01 deg; joints [26.212, -43.795, 101.694, -150.007, 62.127, 165.974]
  MoveL 3432 to (-324.6, -16.81, -30) mm, rotated rx 180 ry 0 rz 0.01 deg; joints [26.34, -43.81, 101.72, -149.87, 62.171, 165.913]
  MoveL 3433 to (-324.44, -16.49, -30) mm, rotated rx 180 ry 0 rz 0.01 deg; joints [26.354, -43.81, 101.721, -149.856, 62.175, 165.907]
  MoveL 3434 to (-322.84, -13.04, -30) mm, rotated rx 180 ry 0 rz 0.01 deg; joints [26.497, -43.809, 101.711, -149.697, 62.206, 165.828]
  MoveL 3435 to (-322.72, -12.74, -30) mm, rotated rx 180 ry 0 rz 0.01 deg; joints [26.509, -43.808, 101.709, -149.684, 62.208, 165.82]
  MoveL 3436 to (-321.51, -9.3, -30) mm, rotated rx 180 ry 0 rz 0.01 deg; joints [26.645, -43.791, 101.666, -149.529, 62.222, 165.735]
  MoveL 3437 to (-321.34, -8.56, -30) mm, rotated rx 180 ry 0 rz 0.01 deg; joints [26.673, -43.784, 101.649, -149.496, 62.221, 165.715]
  MoveL 3438 to (-320.72, -3.12, -30) mm, rotated rx 180 ry 0 rz 0.01 deg; joints [26.866, -43.704, 101.469, -149.259, 62.187, 165.557]
  MoveL 3439 to (-320.7, -2.9, -30) mm, rotated rx -180 ry 0 rz 0.01 deg; joints [26.874, -43.7, 101.46, -149.249, 62.185, 165.551]
  MoveL 3440 to (-320.57, 0.01, -30) mm, rotated rx 180 ry 0 rz 0.01 deg; joints [26.973, -43.649, 101.347, -149.124, 62.159, 165.463]
  MoveL 3441 to (-320.58, 0.42, -30) mm, rotated rx 180 ry 0 rz 0.01 deg; joints [26.987, -43.641, 101.329, -149.107, 62.154, 165.45]
  MoveL 3442 to (-320.74, 2.59, -30) mm, rotated rx -180 ry 0 rz 0.01 deg; joints [27.057, -43.592, 101.221, -149.014, 62.122, 165.379]
  MoveL 3443 to (-320.79, 2.99, -30) mm, rotated rx 180 ry 0 rz 0.01 deg; joints [27.069, -43.582, 101.199, -148.998, 62.116, 165.366]
  MoveL 3444 to (-321.36, 5.89, -30) mm, rotated rx 180 ry 0 rz 0.01 deg; joints [27.156, -43.503, 101.025, -148.877, 62.059, 165.265]
  MoveL 3445 to (-321.49, 6.36, -30) mm, rotated rx -180 ry 0 rz 0.01 deg; joints [27.169, -43.489, 100.994, -148.858, 62.048, 165.248]
  MoveL 3446 to (-322.72, 9.87, -30) mm, rotated rx -180 ry 0 rz 0.01 deg; joints [27.265, -43.371, 100.737, -148.715, 61.955, 165.117]
  MoveL 3447 to (-322.79, 10.06, -30) mm, rotated rx 180 ry 0 rz 0.01 deg; joints [27.27, -43.364, 100.722, -148.708, 61.95, 165.109]
  MoveL 3448 to (-324.35, 13.8, -30) mm, rotated rx 180 ry 0 rz 0.01 deg; joints [27.368, -43.227, 100.425, -148.557, 61.84, 164.964]
  MoveL 3449 to (-324.54, 14.18, -30) mm, rotated rx -180 ry 0 rz 0.01 deg; joints [27.377, -43.212, 100.391, -148.542, 61.828, 164.948]
  MoveL 3450 to (-342.68, 45.66, -30) mm, rotated rx -180 ry 0 rz 0.01 deg; joints [28.094, -41.83, 97.408, -147.293, 60.682, 163.594]
  MoveL 3451 to (-342.91, 46, -30) mm, rotated rx -180 ry 0 rz 0.01 deg; joints [28.101, -41.814, 97.373, -147.28, 60.668, 163.579]
  MoveL 3452 to (-344.86, 48.62, -30) mm, rotated rx -180 ry 0 rz 0.01 deg; joints [28.152, -41.678, 97.081, -147.177, 60.553, 163.454]
  MoveL 3453 to (-344.97, 48.75, -30) mm, rotated rx 180 ry 0 rz 0.01 deg; joints [28.155, -41.67, 97.066, -147.172, 60.547, 163.448]
  MoveL 3454 to (-347.85, 52.23, -30) mm, rotated rx 180 ry 0 rz 0.01 deg; joints [28.216, -41.477, 96.652, -147.036, 60.38, 163.276]
  MoveL 3455 to (-348.15, 52.54, -30) mm, rotated rx 180 ry 0 rz 0.01 deg; joints [28.221, -41.459, 96.612, -147.024, 60.364, 163.26]
  MoveL 3456 to (-350.23, 54.48, -30) mm, rotated rx 180 ry 0 rz 0.01 deg; joints [28.248, -41.33, 96.337, -146.95, 60.25, 163.154]
  MoveL 3457 to (-350.6, 54.78, -30) mm, rotated rx 180 ry 0 rz 0.01 deg; joints [28.251, -41.309, 96.292, -146.939, 60.231, 163.137]
  MoveL 3458 to (-352.52, 56.13, -30) mm, rotated rx 180 ry 0 rz 0.01 deg; joints [28.261, -41.2, 96.059, -146.889, 60.13, 163.054]
  MoveL 3459 to (-352.88, 56.35, -30) mm, rotated rx 180 ry 0 rz 0.01 deg; joints [28.262, -41.18, 96.018, -146.881, 60.112, 163.039]
  MoveL 3460 to (-356.25, 58.14, -30) mm, rotated rx 180 ry 0 rz 0.01 deg; joints [28.261, -41.001, 95.636, -146.818, 59.943, 162.912]
  MoveL 3461 to (-356.49, 58.26, -30) mm, rotated rx -180 ry 0 rz 0.01 deg; joints [28.261, -40.988, 95.609, -146.814, 59.931, 162.903]
  MoveL 3462 to (-360.84, 60.14, -30) mm, rotated rx 180 ry 0 rz 0.01 deg; joints [28.247, -40.764, 95.134, -146.75, 59.716, 162.752]
  MoveL 3463 to (-361.54, 60.36, -30) mm, rotated rx -180 ry 0 rz 0.01 deg; joints [28.241, -40.73, 95.062, -146.744, 59.683, 162.731]
  MoveL 3464 to (-365.17, 61.07, -30) mm, rotated rx 180 ry 0 rz 0.01 deg; joints [28.202, -40.561, 94.706, -146.727, 59.513, 162.634]
  MoveL 3465 to (-365.48, 61.11, -30) mm, rotated rx 180 ry 0 rz 0.01 deg; joints [28.198, -40.547, 94.676, -146.726, 59.499, 162.626]
  MoveL 3466 to (-369.11, 61.47, -30) mm, rotated rx -180 ry 0 rz 0.01 deg; joints [28.148, -40.385, 94.335, -146.723, 59.333, 162.54]
  MoveL 3467 to (-369.5, 61.48, -30) mm, rotated rx 180 ry 0 rz 0.01 deg; joints [28.142, -40.369, 94.299, -146.723, 59.315, 162.532]
  MoveL 3468 to (-373.49, 61.42, -30) mm, rotated rx 180 ry 0 rz 0.01 deg; joints [28.072, -40.2, 93.945, -146.739, 59.137, 162.453]
  MoveL 3469 to (-374.4, 61.28, -30) mm, rotated rx 180 ry 0 rz 0.01 deg; joints [28.053, -40.164, 93.87, -146.748, 59.098, 162.44]
  MoveL 3470 to (-383.59, 58.54, -30) mm, rotated rx -180 ry 0 rz 0.01 deg; joints [27.813, -39.829, 93.171, -146.893, 58.715, 162.346]
  MoveL 3471 to (-383.91, 58.42, -30) mm, rotated rx 180 ry 0 rz 0.01 deg; joints [27.804, -39.818, 93.147, -146.899, 58.702, 162.343]
  MoveL 3472 to (-384.91, 58.01, -30) mm, rotated rx -180 ry 0 rz 0.01 deg; joints [27.774, -39.784, 93.076, -146.919, 58.661, 162.337]
  MoveL 3473 to (-385.72, 57.54, -30) mm, rotated rx 180 ry 0 rz 0.01 deg; joints [27.746, -39.759, 93.025, -146.942, 58.63, 162.337]
  MoveL 3474 to (-393.65, 51.26, -30) mm, rotated rx 180 ry 0 rz 0.01 deg; joints [27.418, -39.551, 92.6, -147.233, 58.341, 162.392]
  MoveL 3475 to (-394.12, 50.81, -30) mm, rotated rx 180 ry 0 rz 0.01 deg; joints [27.396, -39.541, 92.579, -147.254, 58.324, 162.398]
  MoveL 3476 to (-395.23, 49.52, -30) mm, rotated rx -180 ry 0 rz 0.01 deg; joints [27.337, -39.52, 92.538, -147.312, 58.288, 162.42]
  MoveL 3477 to (-395.53, 49.11, -30) mm, rotated rx -180 ry 0 rz 0.01 deg; joints [27.319, -39.516, 92.53, -147.331, 58.279, 162.429]
  MoveL 3478 to (-397.79, 45.48, -30) mm, rotated rx -180 ry 0 rz 0.01 deg; joints [27.168, -39.496, 92.493, -147.494, 58.217, 162.509]
  MoveL 3479 to (-397.83, 45.41, -30) mm, rotated rx 180 ry 0 rz 0.01 deg; joints [27.165, -39.495, 92.493, -147.497, 58.216, 162.51]
  MoveL 3480 to (-401.76, 38.77, -30) mm, rotated rx -180 ry 0 rz 0.01 deg; joints [26.892, -39.466, 92.442, -147.794, 58.11, 162.661]
  MoveL 3481 to (-401.99, 38.31, -30) mm, rotated rx 180 ry 0 rz 0.01 deg; joints [26.874, -39.466, 92.443, -147.815, 58.105, 162.672]
  MoveL 3482 to (-402.41, 37.28, -30) mm, rotated rx -180 ry 0 rz 0.01 deg; joints [26.835, -39.47, 92.453, -147.86, 58.097, 162.699]
  MoveL 3483 to (-402.55, 36.85, -30) mm, rotated rx 180 ry 0 rz 0.01 deg; joints [26.819, -39.473, 92.46, -147.879, 58.096, 162.711]
  MoveL 3484 to (-403.55, 32.92, -30) mm, rotated rx 180 ry 0 rz 0.01 deg; joints [26.678, -39.512, 92.55, -148.053, 58.094, 162.827]
  MoveL 3485 to (-403.56, 32.86, -30) mm, rotated rx 180 ry 0 rz 0.01 deg; joints [26.676, -39.513, 92.551, -148.056, 58.094, 162.829]
  MoveL 3486 to (-403.78, 31.95, -30) mm, rotated rx -180 ry 0 rz 0.01 deg; joints [26.644, -39.523, 92.573, -148.096, 58.094, 162.856]
  MoveL 3487 to (-403.79, 333.8, -30) mm, rotated rx 180 ry 0 rz 0.01 deg; joints [35.408, -31.238, 74.862, -134.523, 54.381, 150.307]
  MoveL 3488 to (-403.73, 334.87, -30) mm, rotated rx -180 ry 0 rz 0.01 deg; joints [35.437, -31.204, 74.789, -134.473, 54.369, 150.255]
  MoveL 3489 to (-403.53, 335.74, -30) mm, rotated rx -180 ry 0 rz 0.01 deg; joints [35.464, -31.183, 74.746, -134.433, 54.367, 150.218]
  MoveL 3490 to (-403.42, 336, -30) mm, rotated rx 180 ry 0 rz 0.01 deg; joints [35.473, -31.18, 74.738, -134.421, 54.369, 150.209]
  MoveL 3491 to (-403.03, 336.5, -29.83) mm, rotated rx -180 ry 0 rz 0.01 deg; joints [35.493, -31.189, 74.742, -134.397, 54.376, 150.192]
  MoveL 3492 to (-402.62, 336.71, -29.37) mm, rotated rx -180 ry 0 rz 0.01 deg; joints [35.506, -31.222, 74.771, -134.382, 54.38, 150.18]
  MoveL 3493 to (-402.46, 336.75, -28.73) mm, rotated rx -180 ry 0 rz 0.01 deg; joints [35.51, -31.256, 74.788, -134.369, 54.37, 150.163]
  Set speed (500.0 mm/s)
  MoveL 3494 to (-402.46, 336.75, 11) mm, rotated rx 180 ry 0 rz 0.01 deg; joints [35.493, -32.912, 74.899, -133.574, 53.288, 148.796]
  Set speed (500.0 mm/s)
  MoveL 3495 to (-212.83, 109.48, 11) mm, rotated rx 180 ry 0 rz 0.01 deg; joints [32.602, -47.591, 105.129, -143.045, 63.709, 162.554]
  Set speed (500.0 mm/s)
  MoveL 3496 to (-212.83, 109.48, -18.23) mm, rotated rx -180 ry 0 rz 0.01 deg; joints [32.619, -46.087, 105.067, -143.444, 64.869, 163.504]
  Set speed (100.0 mm/s)
  MoveL 3497 to (-212.67, 109.46, -18.85) mm, rotated rx -180 ry 0 rz 0.01 deg; joints [32.622, -46.061, 105.079, -143.451, 64.9, 163.527]
  MoveL 3498 to (-212.22, 109.43, -19.32) mm, rotated rx 180 ry 0 rz 0.01 deg; joints [32.63, -46.054, 105.113, -143.453, 64.936, 163.551]
  MoveL 3499 to (-211.61, 109.45, -19.5) mm, rotated rx 180 ry 0 rz 0.01 deg; joints [32.644, -46.067, 105.16, -143.449, 64.967, 163.567]
  MoveL 3500 to (-206.37, 113.47, -19.74) mm, rotated rx 180 ry 0 rz 0.01 deg; joints [32.884, -46.155, 105.364, -143.229, 65.134, 163.534]
  MoveL 3501 to (-207.96, 119.88, -19.99) mm, rotated rx 180 ry 0 rz 0.01 deg; joints [33.058, -45.937, 104.919, -142.983, 65.006, 163.305]
  MoveL 3502 to (-214.47, 121, -20.23) mm, rotated rx 180 ry 0 rz 0.01 deg; joints [32.958, -45.66, 104.356, -143.007, 64.747, 163.161]
  MoveL 3503 to (-218.1, 115.48, -20.48) mm, rotated rx -180 ry 0 rz 0.01 deg; joints [32.705, -45.64, 104.35, -143.277, 64.679, 163.287]
  MoveL 3504 to (-214.5, 109.94, -20.72) mm, rotated rx 180 ry 0 rz 0.01 deg; joints [32.6, -45.886, 104.906, -143.474, 64.896, 163.539]
  MoveL 3505 to (-207.98, 111.03, -20.96) mm, rotated rx -180 ry 0 rz 0.01 deg; joints [32.771, -46.088, 105.358, -143.364, 65.148, 163.625]
  MoveL 3506 to (-206.36, 117.43, -21.21) mm, rotated rx 180 ry 0 rz 0.01 deg; joints [33.013, -45.989, 105.162, -143.083, 65.145, 163.452]
  MoveL 3507 to (-211.58, 121.48, -21.45) mm, rotated rx 180 ry 0 rz 0.01 deg; joints [33.034, -45.692, 104.553, -142.973, 64.902, 163.235]
  MoveL 3508 to (-217.38, 118.32, -21.7) mm, rotated rx 180 ry 0 rz 0.01 deg; joints [32.812, -45.538, 104.259, -143.168, 64.721, 163.244]
  MoveL 3509 to (-216.81, 111.74, -21.94) mm, rotated rx -180 ry 0 rz 0.01 deg; joints [32.611, -45.696, 104.632, -143.439, 64.831, 163.478]
  MoveL 3510 to (-210.55, 109.62, -22.18) mm, rotated rx -180 ry 0 rz 0.01 deg; joints [32.673, -45.962, 105.223, -143.465, 65.112, 163.664]
  MoveL 3511 to (-206.11, 114.51, -22.43) mm, rotated rx -180 ry 0 rz 0.01 deg; joints [32.924, -46.001, 105.323, -143.218, 65.237, 163.591]
  MoveL 3512 to (-208.8, 120.54, -22.67) mm, rotated rx 180 ry 0 rz 0.01 deg; joints [33.063, -45.752, 104.811, -142.999, 65.069, 163.354]
  MoveL 3513 to (-215.4, 120.49, -22.92) mm, rotated rx 180 ry 0 rz 0.01 deg; joints [32.923, -45.498, 104.299, -143.073, 64.82, 163.247]
  MoveL 3514 to (-218, 114.42, -23.16) mm, rotated rx -180 ry 0 rz 0.01 deg; joints [32.674, -45.528, 104.401, -143.355, 64.799, 163.408]
  MoveL 3515 to (-213.48, 109.6, -23.4) mm, rotated rx 180 ry 0 rz 0.01 deg; joints [32.612, -45.791, 104.992, -143.512, 65.045, 163.652]
  MoveL 3516 to (-207.26, 111.81, -23.65) mm, rotated rx -180 ry 0 rz 0.01 deg; joints [32.814, -45.956, 105.364, -143.358, 65.272, 163.697]
  MoveL 3517 to (-206.79, 118.4, -23.89) mm, rotated rx -180 ry 0 rz 0.01 deg; joints [33.037, -45.81, 105.07, -143.082, 65.221, 163.498]
  MoveL 3518 to (-212.64, 121.47, -24.14) mm, rotated rx 180 ry 0 rz 0.01 deg; joints [33.013, -45.513, 104.46, -143.02, 64.964, 163.302]
  MoveL 3519 to (-217.8, 117.34, -24.38) mm, rotated rx -180 ry 0 rz 0.01 deg; joints [32.773, -45.406, 104.266, -143.247, 64.82, 163.354]
  MoveL 3520 to (-216.08, 110.96, -24.62) mm, rotated rx -180 ry 0 rz 0.01 deg; joints [32.603, -45.601, 104.718, -143.498, 64.974, 163.601]
  MoveL 3521 to (-209.55, 109.98, -24.87) mm, rotated rx 180 ry 0 rz 0.01 deg; joints [32.707, -45.85, 105.273, -143.474, 65.252, 163.755]
  MoveL 3522 to (-206.03, 115.57, -25.11) mm, rotated rx 180 ry 0 rz 0.01 deg; joints [32.962, -45.839, 105.266, -143.207, 65.332, 163.643]
  MoveL 3523 to (-209.75, 121.03, -25.36) mm, rotated rx 180 ry 0 rz 0.01 deg; joints [33.061, -45.566, 104.703, -143.023, 65.13, 163.407]
  MoveL 3524 to (-216.24, 119.82, -25.6) mm, rotated rx -180 ry 0 rz 0.01 deg; joints [32.886, -45.343, 104.258, -143.144, 64.899, 163.339]
  MoveL 3525 to (-217.73, 113.39, -25.85) mm, rotated rx 180 ry 0 rz 0.01 deg; joints [32.648, -45.422, 104.463, -143.43, 64.927, 163.531]
  MoveL 3526 to (-212.43, 109.44, -26.09) mm, rotated rx 180 ry 0 rz 0.01 deg; joints [32.63, -45.693, 105.072, -143.542, 65.193, 163.76]
  MoveL 3527 to (-206.69, 112.72, -26.33) mm, rotated rx -180 ry 0 rz 0.01 deg; joints [32.856, -45.816, 105.353, -143.348, 65.388, 163.763]
  MoveL 3528 to (-207.39, 119.28, -26.58) mm, rotated rx -180 ry 0 rz 0.01 deg; joints [33.054, -45.628, 104.968, -143.086, 65.291, 163.544]
  MoveL 3529 to (-213.69, 121.27, -26.82) mm, rotated rx 180 ry 0 rz 0.01 deg; joints [32.987, -45.34, 104.378, -143.073, 65.029, 163.375]
  MoveL 3530 to (-218.04, 116.3, -27.07) mm, rotated rx 180 ry 0 rz 0.01 deg; joints [32.736, -45.281, 104.288, -143.328, 64.927, 163.468]
  MoveL 3531 to (-215.22, 110.33, -27.31) mm, rotated rx -180 ry 0 rz 0.01 deg; joints [32.601, -45.507, 104.805, -143.55, 65.12, 163.721]
  MoveL 3532 to (-208.62, 110.51, -27.55) mm, rotated rx 180 ry 0 rz 0.01 deg; joints [32.745, -45.731, 105.308, -143.476, 65.387, 163.839]
  MoveL 3533 to (-206.15, 116.63, -27.8) mm, rotated rx 180 ry 0 rz 0.01 deg; joints [32.995, -45.67, 105.193, -143.198, 65.42, 163.691]
  MoveL 3534 to (-210.76, 121.36, -28.04) mm, rotated rx 180 ry 0 rz 0.01 deg; joints [33.051, -45.382, 104.597, -143.055, 65.19, 163.463]
  MoveL 3535 to (-216.94, 119.02, -28.29) mm, rotated rx -180 ry 0 rz 0.01 deg; joints [32.847, -45.196, 104.233, -143.219, 64.984, 163.437]
  MoveL 3536 to (-217.27, 112.42, -28.53) mm, rotated rx 180 ry 0 rz 0.01 deg; joints [32.628, -45.321, 104.536, -143.5, 65.061, 163.654]
  MoveL 3537 to (-211.36, 109.47, -28.77) mm, rotated rx -180 ry 0 rz 0.01 deg; joints [32.655, -45.591, 105.142, -143.563, 65.339, 163.862]
  MoveL 3538 to (-206.29, 113.71, -29.02) mm, rotated rx 180 ry 0 rz 0.01 deg; joints [32.898, -45.667, 105.323, -143.337, 65.497, 163.822]
  MoveL 3539 to (-208.14, 120.05, -29.26) mm, rotated rx 180 ry 0 rz 0.01 deg; joints [33.065, -45.443, 104.861, -143.097, 65.356, 163.591]
  MoveL 3540 to (-214.69, 120.9, -29.51) mm, rotated rx -180 ry 0 rz 0.01 deg; joints [32.955, -45.172, 104.308, -143.134, 65.097, 163.454]
  MoveL 3541 to (-218.09, 115.24, -29.75) mm, rotated rx -180 ry 0 rz 0.01 deg; joints [32.702, -45.164, 104.326, -143.407, 65.041, 163.586]
  MoveL 3542 to (-214.27, 109.85, -29.99) mm, rotated rx 180 ry 0 rz 0.01 deg; joints [32.607, -45.412, 104.892, -143.594, 65.267, 163.837]
  MoveL 3543 to (-207.8, 111.19, -30.24) mm, rotated rx 180 ry 0 rz 0.01 deg; joints [32.786, -45.605, 105.326, -143.472, 65.516, 163.915]
  MoveL 3544 to (-206.44, 117.66, -30.48) mm, rotated rx 180 ry 0 rz 0.01 deg; joints [33.024, -45.495, 105.107, -143.193, 65.499, 163.737]
  MoveL 3545 to (-211.82, 121.49, -30.73) mm, rotated rx 180 ry 0 rz 0.01 deg; joints [33.035, -45.2, 104.496, -143.095, 65.25, 163.524]
  MoveL 3546 to (-217.49, 118.1, -30.97) mm, rotated rx -180 ry 0 rz 0.01 deg; joints [32.808, -45.057, 104.224, -143.297, 65.077, 163.541]
  MoveL 3547 to (-216.66, 111.55, -31.21) mm, rotated rx -180 ry 0 rz 0.01 deg; joints [32.614, -45.223, 104.616, -143.563, 65.2, 163.777]
  MoveL 3548 to (-210.32, 109.69, -31.46) mm, rotated rx -180 ry 0 rz 0.01 deg; joints [32.685, -45.483, 105.201, -143.577, 65.482, 163.958]
  MoveL 3549 to (-206.07, 114.75, -31.7) mm, rotated rx 180 ry 0 rz 0.01 deg; joints [32.938, -45.51, 105.276, -143.325, 65.597, 163.877]
  MoveL 3550 to (-209.01, 120.67, -31.95) mm, rotated rx 180 ry 0 rz 0.01 deg; joints [33.068, -45.257, 104.751, -143.115, 65.418, 163.64]
  MoveL 3551 to (-215.61, 120.35, -32.19) mm, rotated rx 180 ry 0 rz 0.01 deg; joints [32.92, -45.012, 104.253, -143.2, 65.171, 163.539]
  MoveL 3552 to (-217.96, 114.18, -32.43) mm, rotated rx -180 ry 0 rz 0.01 deg; joints [32.672, -45.053, 104.378, -143.483, 65.163, 163.707]
  MoveL 3553 to (-213.25, 109.55, -32.68) mm, rotated rx 180 ry 0 rz 0.01 deg; joints [32.62, -45.316, 104.975, -143.629, 65.416, 163.948]
  MoveL 3554 to (-207.12, 112.01, -32.92) mm, rotated rx 180 ry 0 rz 0.01 deg; joints [32.828, -45.47, 105.327, -143.465, 65.637, 163.985]
  MoveL 3555 to (-206.92, 118.61, -33.17) mm, rotated rx -180 ry 0 rz 0.01 deg; joints [33.046, -45.316, 105.011, -143.192, 65.573, 163.782]
  MoveL 3556 to (-212.89, 121.44, -33.41) mm, rotated rx -180 ry 0 rz 0.01 deg; joints [33.012, -45.022, 104.404, -143.142, 65.312, 163.591]
  MoveL 3557 to (-217.87, 117.11, -33.65) mm, rotated rx 180 ry 0 rz 0.01 deg; joints [32.769, -44.926, 104.233, -143.376, 65.177, 163.65]
  MoveL 3558 to (-215.89, 110.8, -33.9) mm, rotated rx 180 ry 0 rz 0.01 deg; joints [32.607, -45.127, 104.701, -143.62, 65.343, 163.899]
  MoveL 3559 to (-209.33, 110.09, -34.14) mm, rotated rx -180 ry 0 rz 0.01 deg; joints [32.72, -45.369, 105.246, -143.583, 65.621, 164.046]
  MoveL 3560 to (-206.04, 115.82, -34.39) mm, rotated rx -180 ry 0 rz 0.01 deg; joints [32.975, -45.346, 105.213, -143.314, 65.689, 163.927]
  MoveL 3561 to (-209.97, 121.12, -34.63) mm, rotated rx -180 ry 0 rz 0.01 deg; joints [33.064, -45.071, 104.641, -143.14, 65.478, 163.692]
  MoveL 3562 to (-216.41, 119.65, -34.88) mm, rotated rx -180 ry 0 rz 0.01 deg; joints [32.882, -44.858, 104.213, -143.271, 65.251, 163.632]
  MoveL 3563 to (-217.64, 113.16, -35.12) mm, rotated rx -180 ry 0 rz 0.01 deg; joints [32.647, -44.947, 104.442, -143.556, 65.292, 163.829]
  MoveL 3564 to (-212.19, 109.43, -35.36) mm, rotated rx 180 ry 0 rz 0.01 deg; joints [32.64, -45.216, 105.051, -143.656, 65.564, 164.054]
  MoveL 3565 to (-206.59, 112.94, -35.61) mm, rotated rx 180 ry 0 rz 0.01 deg; joints [32.871, -45.327, 105.31, -143.454, 65.751, 164.048]
  MoveL 3566 to (-207.55, 119.47, -35.85) mm, rotated rx -180 ry 0 rz 0.01 deg; joints [33.062, -45.132, 104.906, -143.197, 65.641, 163.827]
  MoveL 3567 to (-213.93, 121.2, -36.1) mm, rotated rx 180 ry 0 rz 0.01 deg; joints [32.985, -44.849, 104.323, -143.196, 65.376, 163.663]
  MoveL 3568 to (-218.07, 116.06, -36.34) mm, rotated rx -180 ry 0 rz 0.01 deg; joints [32.733, -44.802, 104.257, -143.455, 65.285, 163.764]
  MoveL 3569 to (-215.01, 110.2, -36.58) mm, rotated rx -180 ry 0 rz 0.01 deg; joints [32.607, -45.032, 104.787, -143.669, 65.489, 164.017]
  MoveL 3570 to (-208.43, 110.65, -36.83) mm, rotated rx 180 ry 0 rz 0.01 deg; joints [32.759, -45.247, 105.275, -143.583, 65.754, 164.127]
  MoveL 3571 to (-206.2, 116.87, -37.07) mm, rotated rx 180 ry 0 rz 0.01 deg; joints [33.007, -45.175, 105.136, -143.305, 65.774, 163.974]
  MoveL 3572 to (-211, 121.4, -37.32) mm, rotated rx -180 ry 0 rz 0.01 deg; joints [33.053, -44.887, 104.534, -143.172, 65.536, 163.748]
  MoveL 3573 to (-217.08, 118.82, -37.56) mm, rotated rx 180 ry 0 rz 0.01 deg; joints [32.843, -44.712, 104.19, -143.346, 65.337, 163.73]
  MoveL 3574 to (-217.15, 112.21, -37.8) mm, rotated rx 180 ry 0 rz 0.01 deg; joints [32.629, -44.845, 104.515, -143.623, 65.426, 163.951]
  MoveL 3575 to (-211.12, 109.51, -38.05) mm, rotated rx 180 ry 0 rz 0.01 deg; joints [32.666, -45.111, 105.117, -143.674, 65.709, 164.154]
  MoveL 3576 to (-206.23, 113.94, -38.29) mm, rotated rx 180 ry 0 rz 0.01 deg; joints [32.912, -45.175, 105.274, -143.441, 65.856, 164.106]
  MoveL 3577 to (-208.33, 120.2, -38.54) mm, rotated rx 180 ry 0 rz 0.01 deg; joints [33.071, -44.946, 104.796, -143.208, 65.704, 163.873]
  MoveL 3578 to (-214.91, 120.79, -38.78) mm, rotated rx -180 ry 0 rz 0.01 deg; joints [32.952, -44.683, 104.254, -143.257, 65.445, 163.743]
  MoveL 3579 to (-218.08, 114.99, -39.02) mm, rotated rx 180 ry 0 rz 0.01 deg; joints [32.7, -44.685, 104.297, -143.533, 65.401, 163.882]
  MoveL 3580 to (-214.04, 109.77, -39.27) mm, rotated rx -180 ry 0 rz 0.01 deg; joints [32.614, -44.935, 104.871, -143.71, 65.637, 164.131]
  MoveL 3581 to (-207.63, 111.37, -39.51) mm, rotated rx 180 ry 0 rz 0.01 deg; joints [32.8, -45.118, 105.288, -143.578, 65.88, 164.201]
  MoveL 3582 to (-206.54, 117.88, -39.76) mm, rotated rx -180 ry 0 rz 0.01 deg; joints [33.034, -44.999, 105.046, -143.3, 65.851, 164.018]
  MoveL 3583 to (-212.06, 121.5, -40) mm, rotated rx 180 ry 0 rz 0.01 deg; joints [33.035, -44.706, 104.434, -143.213, 65.596, 163.809]
  MoveL 3584 to (-214.19, 121.5, -40) mm, rotated rx 180 ry 0 rz 0.01 deg; joints [32.991, -44.629, 104.268, -143.235, 65.511, 163.77]
  MoveC 3585 to (-216.11, 120.39, -40) mm, rotated rx 180 ry 0 rz 0.01 deg; joints [32.915, -44.584, 104.174, -143.301, 65.449, 163.771] to (-216.11, 118.17, -40) mm, rotated rx -180 ry 0 rz 0.01 deg; joints [32.843, -44.634, 104.286, -143.393, 65.477, 163.844]
  MoveL 3586 to (-214.88, 116.02, -40) mm, rotated rx 180 ry 0 rz 0.01 deg; joints [32.8, -44.727, 104.49, -143.469, 65.553, 163.936]
  MoveC 3587 to (-213.84, 114.98, -40) mm, rotated rx -180 ry 0 rz 0.01 deg; joints [32.788, -44.788, 104.623, -143.501, 65.608, 163.988] to (-212.42, 114.6, -40) mm, rotated rx 180 ry 0 rz 0.01 deg; joints [32.805, -44.848, 104.753, -143.501, 65.669, 164.026]
  MoveL 3588 to (-181.08, 114.6, -40) mm, rotated rx -180 ry 0 rz 0.01 deg; joints [33.47, -45.96, 107.157, -143.146, 66.899, 164.582]
  MoveC 3589 to (-179.66, 114.98, -40) mm, rotated rx -180 ry 0 rz 0.01 deg; joints [33.513, -46.002, 107.245, -143.113, 66.95, 164.595] to (-178.62, 116.02, -40) mm, rotated rx -180 ry 0 rz 0.01 deg; joints [33.57, -46.015, 107.271, -143.058, 66.977, 164.58]
  MoveL 3590 to (-177.39, 118.16, -40) mm, rotated rx 180 ry 0 rz 0.01 deg; joints [33.666, -46.01, 107.258, -142.955, 66.997, 164.534]
  MoveC 3591 to (-177.38, 120.39, -40) mm, rotated rx -180 ry 0 rz 0.01 deg; joints [33.739, -45.961, 107.146, -142.864, 66.969, 164.463] to (-179.31, 121.5, -40) mm, rotated rx 180 ry 0 rz 0.01 deg; joints [33.733, -45.869, 106.945, -142.841, 66.88, 164.393]
  MoveL 3592 to (-212.06, 121.5, -40) mm, rotated rx 180 ry 0 rz 0.01 deg; joints [33.035, -44.706, 104.434, -143.213, 65.596, 163.809]
  MoveC 3593 to (-215.5, 122.55, -40) mm, rotated rx -180 ry 0 rz 0.01 deg; joints [32.997, -44.557, 104.113, -143.206, 65.446, 163.712] to (-217.77, 125.34, -40) mm, rotated rx 180 ry 0 rz 0.01 deg; joints [33.039, -44.412, 103.795, -143.114, 65.321, 163.579]
  MoveC 3594 to (-219.94, 128.17, -40) mm, rotated rx 180 ry 0 rz 0.01 deg; joints [33.085, -44.268, 103.481, -143.019, 65.198, 163.446] to (-223.25, 129.5, -40) mm, rotated rx -180 ry 0 rz 0.01 deg; joints [33.058, -44.117, 103.154, -142.998, 65.05, 163.341]
  MoveC 3595 to (-226.52, 129.87, -40) mm, rotated rx -180 ry 0 rz 0.01 deg; joints [33.002, -43.989, 102.878, -143.015, 64.914, 163.269] to (-229.79, 130.22, -40) mm, rotated rx 180 ry 0 rz 0.01 deg; joints [32.946, -43.861, 102.602, -143.032, 64.779, 163.196]
  MoveC 3596 to (-231.58, 129.31, -40) mm, rotated rx 180 ry 0 rz 0.01 deg; joints [32.88, -43.816, 102.506, -143.088, 64.718, 163.193] to (-231.48, 127.29, -40) mm, rotated rx -180 ry 0 rz 0.01 deg; joints [32.818, -43.866, 102.618, -143.17, 64.748, 163.262]
  MoveC 3597 to (-228.69, 123.32, -40) mm, rotated rx -180 ry 0 rz 0.01 deg; joints [32.749, -44.059, 103.039, -143.307, 64.909, 163.445] to (-226.06, 119.24, -40) mm, rotated rx 180 ry 0 rz 0.01 deg; joints [32.672, -44.248, 103.453, -143.45, 65.066, 163.628]
  MoveC 3598 to (-223.54, 115.1, -40) mm, rotated rx 180 ry 0 rz 0.01 deg; joints [32.591, -44.433, 103.859, -143.596, 65.219, 163.809] to (-221.09, 110.91, -40) mm, rotated rx -180 ry 0 rz 0.01 deg; joints [32.506, -44.616, 104.26, -143.745, 65.37, 163.99]
  MoveC 3599 to (-217.99, 107.8, -40) mm, rotated rx 180 ry 0 rz 0.01 deg; joints [32.47, -44.798, 104.658, -143.841, 65.533, 164.146] to (-213.74, 106.66, -40) mm, rotated rx 180 ry 0 rz 0.01 deg; joints [32.52, -44.976, 105.045, -143.844, 65.716, 164.258]
  MoveL 3600 to (-179.77, 106.66, -40) mm, rotated rx -180 ry 0 rz 0.01 deg; joints [33.238, -46.181, 107.65, -143.457, 67.052, 164.856]
  MoveC 3601 to (-175.52, 107.8, -40) mm, rotated rx 180 ry 0 rz 0.01 deg; joints [33.368, -46.304, 107.915, -143.358, 67.202, 164.894] to (-172.41, 110.91, -40) mm, rotated rx 180 ry 0 rz 0.01 deg; joints [33.537, -46.344, 107.995, -143.191, 67.283, 164.85]
  MoveC 3602 to (-169.96, 115.09, -40) mm, rotated rx -180 ry 0 rz 0.01 deg; joints [33.728, -46.336, 107.97, -142.989, 67.324, 164.761] to (-167.45, 119.23, -40) mm, rotated rx 180 ry 0 rz 0.01 deg; joints [33.918, -46.331, 107.951, -142.788, 67.367, 164.673]
  MoveC 3603 to (-164.84, 123.31, -40) mm, rotated rx -180 ry 0 rz 0.01 deg; joints [34.109, -46.33, 107.941, -142.588, 67.415, 164.589] to (-162.07, 127.29, -40) mm, rotated rx -180 ry 0 rz 0.01 deg; joints [34.3, -46.336, 107.946, -142.39, 67.47, 164.511]
  MoveC 3604 to (-161.96, 129.3, -40) mm, rotated rx 180 ry 0 rz 0.01 deg; joints [34.368, -46.294, 107.852, -142.306, 67.448, 164.448] to (-163.76, 130.22, -40) mm, rotated rx 180 ry 0 rz 0.01 deg; joints [34.358, -46.211, 107.671, -142.292, 67.367, 164.388]
  MoveC 3605 to (-167.47, 129.82, -40) mm, rotated rx -180 ry 0 rz 0.01 deg; joints [34.263, -46.093, 107.414, -142.355, 67.23, 164.335] to (-171.17, 129.4, -40) mm, rotated rx -180 ry 0 rz 0.01 deg; joints [34.167, -45.974, 107.158, -142.418, 67.093, 164.283]
  MoveC 3606 to (-174.89, 129.08, -40) mm, rotated rx 180 ry 0 rz 0.01 deg; joints [34.075, -45.852, 106.894, -142.477, 66.954, 164.228] to (-178.62, 128.97, -40) mm, rotated rx -180 ry 0 rz 0.01 deg; joints [33.991, -45.724, 106.619, -142.527, 66.811, 164.166]
  MoveL 3607 to (-214.9, 128.97, -40) mm, rotated rx -180 ry 0 rz 0.01 deg; joints [33.215, -44.433, 103.834, -142.935, 65.389, 163.512]
  MoveC 3608 to (-218.63, 129.08, -40) mm, rotated rx -180 ry 0 rz 0.01 deg; joints [33.141, -44.295, 103.537, -142.969, 65.239, 163.44] to (-222.36, 129.4, -40) mm, rotated rx -180 ry 0 rz 0.01 deg; joints [33.073, -44.152, 103.229, -142.993, 65.087, 163.361]
  MoveL 3609 to (-223.25, 129.5, -40) mm, rotated rx 180 ry 0 rz 0.01 deg; joints [33.058, -44.117, 103.154, -142.998, 65.05, 163.341]
  MoveC 3610 to (-226.42, 130.85, -40) mm, rotated rx 180 ry 0 rz 0.01 deg; joints [33.036, -43.97, 102.835, -142.973, 64.906, 163.238] to (-228.33, 133.72, -40) mm, rotated rx 180 ry 0 rz 0.01 deg; joints [33.087, -43.834, 102.537, -142.874, 64.793, 163.107]
  MoveC 3611 to (-230.25, 136.58, -40) mm, rotated rx -180 ry 0 rz 0.01 deg; joints [33.138, -43.697, 102.239, -142.774, 64.68, 162.975] to (-233.42, 137.94, -40) mm, rotated rx -180 ry 0 rz 0.01 deg; joints [33.116, -43.548, 101.918, -142.748, 64.536, 162.87]
  MoveC 3612 to (-237.03, 138.38, -40) mm, rotated rx 180 ry 0 rz 0.01 deg; joints [33.055, -43.404, 101.608, -142.763, 64.385, 162.787] to (-240.64, 138.86, -40) mm, rotated rx 180 ry 0 rz 0.01 deg; joints [32.997, -43.259, 101.295, -142.777, 64.233, 162.702]
  MoveC 3613 to (-242.32, 139.13, -40) mm, rotated rx -180 ry 0 rz 0.01 deg; joints [32.971, -43.189, 101.147, -142.781, 64.162, 162.661] to (-243.99, 139.48, -40) mm, rotated rx 180 ry 0 rz 0.01 deg; joints [32.948, -43.119, 100.996, -142.781, 64.09, 162.617]
  MoveC 3614 to (-245.65, 139.85, -40) mm, rotated rx -180 ry 0 rz 0.01 deg; joints [32.925, -43.048, 100.844, -142.781, 64.018, 162.573] to (-247.32, 140.18, -40) mm, rotated rx 180 ry 0 rz 0.01 deg; joints [32.902, -42.978, 100.693, -142.781, 63.946, 162.53]
  MoveC 3615 to (-249.04, 139.39, -40) mm, rotated rx -180 ry 0 rz 0.01 deg; joints [32.843, -42.932, 100.595, -142.829, 63.886, 162.524] to (-248.85, 137.51, -40) mm, rotated rx -180 ry 0 rz 0.01 deg; joints [32.787, -42.983, 100.707, -142.906, 63.917, 162.591]
  MoveL 3616 to (-243.27, 131.12, -40) mm, rotated rx -180 ry 0 rz 0.01 deg; joints [32.699, -43.34, 101.485, -143.121, 64.224, 162.913]
  MoveC 3617 to (-240.52, 127.87, -40) mm, rotated rx 180 ry 0 rz 0.01 deg; joints [32.652, -43.517, 101.869, -143.231, 64.375, 163.074] to (-237.91, 124.52, -40) mm, rotated rx -180 ry 0 rz 0.01 deg; joints [32.598, -43.691, 102.248, -143.346, 64.523, 163.234]
  MoveC 3618 to (-234.43, 119.5, -40) mm, rotated rx -180 ry 0 rz 0.01 deg; joints [32.509, -43.934, 102.779, -143.521, 64.727, 163.465] to (-231.31, 114.23, -40) mm, rotated rx -180 ry 0 rz 0.01 deg; joints [32.404, -44.168, 103.29, -143.709, 64.918, 163.696]
  MoveC 3619 to (-228.36, 108.88, -40) mm, rotated rx -180 ry 0 rz 0.01 deg; joints [32.291, -44.396, 103.79, -143.902, 65.104, 163.924] to (-225.34, 103.56, -40) mm, rotated rx -180 ry 0 rz 0.01 deg; joints [32.181, -44.624, 104.291, -144.092, 65.291, 164.151]
  MoveC 3620 to (-222.23, 100.45, -40) mm, rotated rx -180 ry 0 rz 0.01 deg; joints [32.143, -44.806, 104.688, -144.19, 65.455, 164.306] to (-217.99, 99.31, -40) mm, rotated rx -180 ry 0 rz 0.01 deg; joints [32.193, -44.984, 105.076, -144.193, 65.639, 164.418]
  MoveL 3621 to (-175.53, 99.31, -40) mm, rotated rx 180 ry 0 rz 0.01 deg; joints [33.087, -46.489, 108.333, -143.707, 67.31, 165.16]
  MoveC 3622 to (-171.28, 100.45, -40) mm, rotated rx 180 ry 0 rz 0.01 deg; joints [33.217, -46.612, 108.597, -143.607, 67.46, 165.197] to (-168.17, 103.56, -40) mm, rotated rx -180 ry 0 rz 0.01 deg; joints [33.387, -46.652, 108.677, -143.44, 67.541, 165.154]
  MoveC 3623 to (-167.08, 105.51, -40) mm, rotated rx -180 ry 0 rz 0.01 deg; joints [33.476, -46.647, 108.662, -143.346, 67.558, 165.112] to (-166.05, 107.49, -40) mm, rotated rx 180 ry 0 rz 0.01 deg; joints [33.563, -46.638, 108.641, -143.252, 67.572, 165.067]
  MoveC 3624 to (-165.03, 109.48, -40) mm, rotated rx 180 ry 0 rz 0.01 deg; joints [33.651, -46.63, 108.619, -143.157, 67.585, 165.023] to (-163.94, 111.43, -40) mm, rotated rx 180 ry 0 rz 0.01 deg; joints [33.739, -46.625, 108.603, -143.063, 67.602, 164.98]
  MoveC 3625 to (-159.65, 118.33, -40) mm, rotated rx 180 ry 0 rz 0.01 deg; joints [34.061, -46.619, 108.578, -142.725, 67.678, 164.837] to (-154.93, 124.94, -40) mm, rotated rx 180 ry 0 rz 0.01 deg; joints [34.382, -46.633, 108.596, -142.393, 67.772, 164.71]
  MoveC 3626 to (-149.89, 131.31, -40) mm, rotated rx 180 ry 0 rz 0.01 deg; joints [34.703, -46.661, 108.644, -142.066, 67.881, 164.595] to (-144.65, 137.52, -40) mm, rotated rx 180 ry 0 rz 0.01 deg; joints [35.024, -46.697, 108.712, -141.743, 67.998, 164.488]
  MoveC 3627 to (-144.47, 139.39, -40) mm, rotated rx -180 ry 0 rz 0.01 deg; joints [35.089, -46.661, 108.629, -141.664, 67.981, 164.431] to (-146.19, 140.18, -40) mm, rotated rx 180 ry 0 rz 0.01 deg; joints [35.075, -46.585, 108.462, -141.655, 67.906, 164.376]
  MoveC 3628 to (-169.67, 136.82, -40) mm, rotated rx -180 ry 0 rz 0.01 deg; joints [34.44, -45.857, 106.891, -142.096, 67.055, 164.071] to (-193.36, 135.65, -40) mm, rotated rx 180 ry 0 rz 0.01 deg; joints [33.886, -45.053, 105.156, -142.426, 66.152, 163.685]
  MoveC 3629 to (-213.42, 136.2, -40) mm, rotated rx 180 ry 0 rz 0.01 deg; joints [33.477, -44.321, 103.579, -142.621, 65.356, 163.301] to (-233.42, 137.94, -40) mm, rotated rx -180 ry 0 rz 0.01 deg; joints [33.116, -43.548, 101.918, -142.748, 64.536, 162.87]
  MoveC 3630 to (-236.18, 139.16, -40) mm, rotated rx 180 ry 0 rz 0.01 deg; joints [33.097, -43.417, 101.635, -142.723, 64.409, 162.777] to (-237.78, 141.72, -40) mm, rotated rx -180 ry 0 rz 0.01 deg; joints [33.145, -43.298, 101.375, -142.632, 64.313, 162.66]
  MoveC 3631 to (-239.32, 144.3, -40) mm, rotated rx -180 ry 0 rz 0.01 deg; joints [33.195, -43.18, 101.119, -142.539, 64.218, 162.543] to (-241.99, 145.67, -40) mm, rotated rx -180 ry 0 rz 0.01 deg; joints [33.183, -43.048, 100.834, -142.507, 64.093, 162.445]
  MoveC 3632 to (-243.73, 146.02, -40) mm, rotated rx 180 ry 0 rz 0.01 deg; joints [33.158, -42.975, 100.677, -142.508, 64.018, 162.4] to (-245.46, 146.39, -40) mm, rotated rx 180 ry 0 rz 0.01 deg; joints [33.134, -42.902, 100.518, -142.508, 63.944, 162.354]
  MoveC 3633 to (-260.32, 150.37, -40) mm, rotated rx 180 ry 0 rz 0.01 deg; joints [32.957, -42.244, 99.108, -142.467, 63.288, 161.927] to (-274.77, 155.67, -40) mm, rotated rx 180 ry 0 rz 0.01 deg; joints [32.832, -41.561, 97.643, -142.356, 62.626, 161.453]
  MoveC 3634 to (-276.33, 155.15, -40) mm, rotated rx -180 ry 0 rz 0.01 deg; joints [32.785, -41.513, 97.542, -142.389, 62.568, 161.44] to (-276, 153.54, -40) mm, rotated rx -180 ry 0 rz 0.01 deg; joints [32.742, -41.565, 97.655, -142.454, 62.602, 161.503]
  MoveC 3635 to (-266.96, 146.17, -40) mm, rotated rx -180 ry 0 rz 0.01 deg; joints [32.694, -42.09, 98.787, -142.694, 63.067, 161.941] to (-258.51, 138.15, -40) mm, rotated rx -180 ry 0 rz 0.01 deg; joints [32.613, -42.603, 99.894, -142.961, 63.515, 162.383]
  MoveC 3636 to (-250.64, 129.55, -40) mm, rotated rx 180 ry 0 rz 0.01 deg; joints [32.5, -43.1, 100.973, -143.252, 63.944, 162.826] to (-243.36, 120.45, -40) mm, rotated rx 180 ry 0 rz 0.01 deg; joints [32.358, -43.581, 102.02, -143.565, 64.353, 163.268]
  MoveC 3637 to (-241.14, 117.36, -40) mm, rotated rx -180 ry 0 rz 0.01 deg; joints [32.304, -43.734, 102.353, -143.673, 64.482, 163.412] to (-239.05, 114.17, -40) mm, rotated rx -180 ry 0 rz 0.01 deg; joints [32.245, -43.884, 102.68, -143.786, 64.606, 163.556]
  MoveC 3638 to (-237.05, 110.93, -40) mm, rotated rx -180 ry 0 rz 0.01 deg; joints [32.181, -44.03, 103.001, -143.901, 64.728, 163.699] to (-235.12, 107.65, -40) mm, rotated rx 180 ry 0 rz 0.01 deg; joints [32.115, -44.175, 103.318, -144.019, 64.847, 163.841]
  MoveC 3639 to (-233.61, 104.95, -40) mm, rotated rx 180 ry 0 rz 0.01 deg; joints [32.058, -44.29, 103.57, -144.117, 64.941, 163.956] to (-232.2, 102.2, -40) mm, rotated rx -180 ry 0 rz 0.01 deg; joints [31.997, -44.403, 103.818, -144.217, 65.033, 164.071]
  MoveC 3640 to (-230.78, 99.45, -40) mm, rotated rx -180 ry 0 rz 0.01 deg; joints [31.937, -44.516, 104.065, -144.318, 65.124, 164.185] to (-229.28, 96.75, -40) mm, rotated rx -180 ry 0 rz 0.01 deg; joints [31.879, -44.63, 104.316, -144.415, 65.218, 164.299]
  MoveC 3641 to (-226.17, 93.64, -40) mm, rotated rx -180 ry 0 rz 0.01 deg; joints [31.841, -44.811, 104.713, -144.513, 65.382, 164.454] to (-221.93, 92.5, -40) mm, rotated rx 180 ry 0 rz 0.01 deg; joints [31.89, -44.99, 105.101, -144.517, 65.566, 164.566]
  MoveL 3642 to (-171.59, 92.5, -40) mm, rotated rx 180 ry 0 rz 0.01 deg; joints [32.946, -46.772, 108.961, -143.939, 67.55, 165.439]
  MoveC 3643 to (-167.35, 93.64, -40) mm, rotated rx 180 ry 0 rz 0.01 deg; joints [33.076, -46.895, 109.224, -143.838, 67.7, 165.476] to (-164.23, 96.75, -40) mm, rotated rx -180 ry 0 rz 0.01 deg; joints [33.247, -46.935, 109.305, -143.67, 67.78, 165.433]
  MoveC 3644 to (-162.67, 99.56, -40) mm, rotated rx 180 ry 0 rz 0.01 deg; joints [33.375, -46.928, 109.285, -143.534, 67.804, 165.373] to (-161.19, 102.41, -40) mm, rotated rx -180 ry 0 rz 0.01 deg; joints [33.502, -46.916, 109.254, -143.398, 67.824, 165.309]
  MoveC 3645 to (-159.71, 105.27, -40) mm, rotated rx 180 ry 0 rz 0.01 deg; joints [33.629, -46.905, 109.224, -143.261, 67.844, 165.246] to (-158.15, 108.08, -40) mm, rotated rx 180 ry 0 rz 0.01 deg; joints [33.757, -46.897, 109.201, -143.125, 67.867, 165.185]
  MoveC 3646 to (-149.77, 120.95, -40) mm, rotated rx -180 ry 0 rz 0.01 deg; joints [34.367, -46.898, 109.178, -142.487, 68.02, 164.925] to (-140.06, 132.85, -40) mm, rotated rx 180 ry 0 rz 0.01 deg; joints [34.977, -46.958, 109.287, -141.87, 68.232, 164.717]
  MoveC 3647 to (-129.23, 143.73, -40) mm, rotated rx 180 ry 0 rz 0.01 deg; joints [35.58, -47.073, 109.516, -141.277, 68.496, 164.557] to (-117.46, 153.58, -40) mm, rotated rx 180 ry 0 rz 0.01 deg; joints [36.174, -47.236, 109.853, -140.709, 68.803, 164.446]
  MoveC 3648 to (-117.14, 155.19, -40) mm, rotated rx -180 ry 0 rz 0.01 deg; joints [36.233, -47.209, 109.792, -140.64, 68.794, 164.4] to (-118.69, 155.7, -40) mm, rotated rx -180 ry 0 rz 0.01 deg; joints [36.213, -47.146, 109.653, -140.642, 68.729, 164.356]
  MoveC 3649 to (-128.96, 151.77, -40) mm, rotated rx 180 ry 0 rz 0.01 deg; joints [35.846, -46.897, 109.118, -140.948, 68.4, 164.304] to (-139.48, 148.59, -40) mm, rotated rx 180 ry 0 rz 0.01 deg; joints [35.5, -46.618, 108.518, -141.223, 68.049, 164.223]
  MoveC 3650 to (-150.18, 146.11, -40) mm, rotated rx 180 ry 0 rz 0.01 deg; joints [35.176, -46.313, 107.861, -141.468, 67.678, 164.114] to (-161.02, 144.28, -40) mm, rotated rx 180 ry 0 rz 0.01 deg; joints [34.873, -45.984, 107.153, -141.684, 67.29, 163.982]
  MoveC 3651 to (-169.8, 143.36, -40) mm, rotated rx -180 ry 0 rz 0.01 deg; joints [34.648, -45.702, 106.544, -141.831, 66.966, 163.856] to (-178.62, 143.06, -40) mm, rotated rx -180 ry 0 rz 0.01 deg; joints [34.444, -45.402, 105.896, -141.951, 66.63, 163.708]
  MoveL 3652 to (-214.9, 143.06, -40) mm, rotated rx 180 ry 0 rz 0.01 deg; joints [33.663, -44.108, 103.11, -142.354, 65.211, 163.045]
  MoveC 3653 to (-228.51, 143.71, -40) mm, rotated rx 180 ry 0 rz 0.01 deg; joints [33.399, -43.595, 102.007, -142.463, 64.66, 162.768] to (-241.99, 145.67, -40) mm, rotated rx -180 ry 0 rz 0.01 deg; joints [33.183, -43.048, 100.834, -142.507, 64.093, 162.445]
  MoveC 3654 to (-244.74, 147.12, -40) mm, rotated rx 180 ry 0 rz 0.01 deg; joints [33.172, -42.911, 100.537, -142.471, 63.964, 162.343] to (-246.22, 149.86, -40) mm, rotated rx -180 ry 0 rz 0.01 deg; joints [33.227, -42.791, 100.276, -142.371, 63.869, 162.22]
  MoveC 3655 to (-247.65, 152.61, -40) mm, rotated rx 180 ry 0 rz 0.01 deg; joints [33.284, -42.671, 100.016, -142.269, 63.777, 162.098] to (-250.33, 154.16, -40) mm, rotated rx 180 ry 0 rz 0.01 deg; joints [33.277, -42.533, 99.717, -142.228, 63.648, 161.992]
  MoveC 3656 to (-257.55, 156.1, -40) mm, rotated rx 180 ry 0 rz 0.01 deg; joints [33.191, -42.213, 99.031, -142.207, 63.33, 161.782] to (-264.67, 158.35, -40) mm, rotated rx -180 ry 0 rz 0.01 deg; joints [33.117, -41.886, 98.331, -142.169, 63.01, 161.562]
  MoveC 3657 to (-269.26, 160.1, -40) mm, rotated rx 180 ry 0 rz 0.01 deg; joints [33.078, -41.667, 97.861, -142.131, 62.799, 161.408] to (-273.71, 162.17, -40) mm, rotated rx -180 ry 0 rz 0.01 deg; joints [33.053, -41.444, 97.383, -142.077, 62.589, 161.244]
  MoveL 3658 to (-283.28, 167.03, -40) mm, rotated rx -180 ry 0 rz 0.01 deg; joints [33.011, -40.951, 96.327, -141.939, 62.131, 160.874]
  MoveC 3659 to (-285.54, 166.94, -40) mm, rotated rx 180 ry 0 rz 0.01 deg; joints [32.964, -40.864, 96.142, -141.958, 62.037, 160.83] to (-286.65, 164.96, -40) mm, rotated rx -180 ry 0 rz 0.01 deg; joints [32.882, -40.869, 96.157, -142.048, 62.015, 160.878]
  MoveL 3660 to (-286.65, 156.54, -40) mm, rotated rx -180 ry 0 rz 0.01 deg; joints [32.624, -41.076, 96.609, -142.401, 62.121, 161.179]
  MoveC 3661 to (-285.88, 153.39, -40) mm, rotated rx 180 ry 0 rz 0.01 deg; joints [32.543, -41.182, 96.841, -142.528, 62.192, 161.307] to (-283.75, 150.96, -40) mm, rotated rx 180 ry 0 rz 0.01 deg; joints [32.51, -41.325, 97.148, -142.616, 62.311, 161.437]
  MoveC 3662 to (-271.17, 141.13, -40) mm, rotated rx -180 ry 0 rz 0.01 deg; joints [32.454, -42.048, 98.705, -142.936, 62.956, 162.033] to (-259.7, 130.04, -40) mm, rotated rx -180 ry 0 rz 0.01 deg; joints [32.334, -42.747, 100.216, -143.308, 63.567, 162.637]
  MoveC 3663 to (-249.5, 117.75, -40) mm, rotated rx -180 ry 0 rz 0.01 deg; joints [32.149, -43.413, 101.664, -143.732, 64.137, 163.243] to (-240.76, 104.4, -40) mm, rotated rx 180 ry 0 rz 0.01 deg; joints [31.896, -44.038, 103.03, -144.208, 64.659, 163.844]
  MoveC 3664 to (-238.79, 100.85, -40) mm, rotated rx 180 ry 0 rz 0.01 deg; joints [31.821, -44.19, 103.362, -144.337, 64.782, 163.995] to (-236.94, 97.25, -40) mm, rotated rx 180 ry 0 rz 0.01 deg; joints [31.741, -44.337, 103.686, -144.469, 64.902, 164.145]
  MoveC 3665 to (-235.08, 93.65, -40) mm, rotated rx -180 ry 0 rz 0.01 deg; joints [31.662, -44.484, 104.009, -144.601, 65.022, 164.294] to (-233.11, 90.11, -40) mm, rotated rx -180 ry 0 rz 0.01 deg; joints [31.586, -44.634, 104.337, -144.729, 65.146, 164.443]
  MoveC 3666 to (-230.01, 87, -40) mm, rotated rx 180 ry 0 rz 0.01 deg; joints [31.546, -44.814, 104.733, -144.828, 65.31, 164.597] to (-225.76, 85.86, -40) mm, rotated rx 180 ry 0 rz 0.01 deg; joints [31.595, -44.994, 105.122, -144.832, 65.495, 164.708]
  MoveL 3667 to (-167.77, 85.86, -40) mm, rotated rx 180 ry 0 rz 0.01 deg; joints [32.807, -47.046, 109.57, -144.165, 67.783, 165.708]
  MoveC 3668 to (-163.52, 87, -40) mm, rotated rx 180 ry 0 rz 0.01 deg; joints [32.937, -47.168, 109.832, -144.063, 67.933, 165.745] to (-160.4, 90.11, -40) mm, rotated rx 180 ry 0 rz 0.01 deg; joints [33.109, -47.208, 109.914, -143.894, 68.013, 165.702]
  MoveC 3669 to (-158.37, 93.76, -40) mm, rotated rx 180 ry 0 rz 0.01 deg; joints [33.276, -47.199, 109.888, -143.717, 68.044, 165.624] to (-156.46, 97.46, -40) mm, rotated rx -180 ry 0 rz 0.01 deg; joints [33.442, -47.185, 109.849, -143.539, 68.069, 165.543]
  MoveC 3670 to (-154.54, 101.17, -40) mm, rotated rx -180 ry 0 rz 0.01 deg; joints [33.607, -47.17, 109.81, -143.361, 68.095, 165.461] to (-152.51, 104.82, -40) mm, rotated rx 180 ry 0 rz 0.01 deg; joints [33.774, -47.16, 109.78, -143.184, 68.125, 165.383]
  MoveC 3671 to (-143.8, 118.07, -40) mm, rotated rx -180 ry 0 rz 0.01 deg; joints [34.407, -47.163, 109.762, -142.524, 68.284, 165.118] to (-133.65, 130.23, -40) mm, rotated rx 180 ry 0 rz 0.01 deg; joints [35.038, -47.232, 109.889, -141.887, 68.508, 164.91]
  MoveC 3672 to (-122.23, 141.23, -40) mm, rotated rx -180 ry 0 rz 0.01 deg; joints [35.661, -47.362, 110.152, -141.278, 68.789, 164.758] to (-109.75, 150.99, -40) mm, rotated rx 180 ry 0 rz 0.01 deg; joints [36.273, -47.549, 110.54, -140.699, 69.121, 164.662]
  MoveC 3673 to (-107.63, 153.42, -40) mm, rotated rx 180 ry 0 rz 0.01 deg; joints [36.402, -47.562, 110.564, -140.569, 69.167, 164.621] to (-106.86, 156.56, -40) mm, rotated rx 180 ry 0 rz 0.01 deg; joints [36.522, -47.514, 110.454, -140.431, 69.153, 164.534]
  MoveL 3674 to (-106.86, 164.94, -40) mm, rotated rx -180 ry 0 rz 0.01 deg; joints [36.791, -47.318, 110.011, -140.095, 69.042, 164.264]
  MoveC 3675 to (-107.97, 166.91, -40) mm, rotated rx 180 ry 0 rz 0.01 deg; joints [36.828, -47.235, 109.827, -140.033, 68.975, 164.18] to (-110.23, 166.99, -40) mm, rotated rx 180 ry 0 rz 0.01 deg; joints [36.776, -47.159, 109.662, -140.063, 68.891, 164.138]
  MoveC 3676 to (-122.58, 161.29, -40) mm, rotated rx 180 ry 0 rz 0.01 deg; joints [36.301, -46.886, 109.078, -140.473, 68.512, 164.107] to (-135.4, 156.72, -40) mm, rotated rx -180 ry 0 rz 0.01 deg; joints [35.856, -46.566, 108.39, -140.838, 68.095, 164.031]
  MoveC 3677 to (-148.55, 153.26, -40) mm, rotated rx -180 ry 0 rz 0.01 deg; joints [35.442, -46.202, 107.609, -141.157, 67.646, 163.911] to (-161.93, 150.85, -40) mm, rotated rx 180 ry 0 rz 0.01 deg; joints [35.063, -45.8, 106.743, -141.428, 67.17, 163.752]
  MoveC 3678 to (-170.26, 149.98, -40) mm, rotated rx 180 ry 0 rz 0.01 deg; joints [34.849, -45.533, 106.166, -141.567, 66.863, 163.631] to (-178.62, 149.69, -40) mm, rotated rx -180 ry 0 rz 0.01 deg; joints [34.655, -45.248, 105.551, -141.68, 66.545, 163.49]
  MoveL 3679 to (-214.9, 149.69, -40) mm, rotated rx 180 ry 0 rz 0.01 deg; joints [33.873, -43.953, 102.764, -142.081, 65.127, 162.822]
  MoveC 3680 to (-227.57, 150.27, -40) mm, rotated rx -180 ry 0 rz 0.01 deg; joints [33.625, -43.475, 101.739, -142.183, 64.615, 162.564] to (-240.14, 151.98, -40) mm, rotated rx -180 ry 0 rz 0.01 deg; joints [33.418, -42.968, 100.651, -142.229, 64.089, 162.265]
  MoveC 3681 to (-245.25, 152.99, -40) mm, rotated rx 180 ry 0 rz 0.01 deg; joints [33.345, -42.753, 100.188, -142.233, 63.869, 162.131] to (-250.33, 154.16, -40) mm, rotated rx 180 ry 0 rz 0.01 deg; joints [33.277, -42.533, 99.717, -142.228, 63.648, 161.992]
  MoveC 3682 to (-253.66, 156.16, -40) mm, rotated rx 180 ry 0 rz 0.01 deg; joints [33.271, -42.359, 99.343, -142.173, 63.488, 161.857] to (-255.28, 159.68, -40) mm, rotated rx -180 ry 0 rz 0.01 deg; joints [33.347, -42.213, 99.024, -142.04, 63.377, 161.702]
  MoveC 3683 to (-256.81, 163.22, -40) mm, rotated rx 180 ry 0 rz 0.01 deg; joints [33.425, -42.069, 98.712, -141.905, 63.271, 161.548] to (-259.96, 165.43, -40) mm, rotated rx 180 ry 0 rz 0.01 deg; joints [33.429, -41.895, 98.336, -141.838, 63.114, 161.407]
  MoveC 3684 to (-276.24, 172.32, -40) mm, rotated rx 180 ry 0 rz 0.01 deg; joints [33.312, -41.096, 96.625, -141.671, 62.357, 160.83] to (-291.51, 181.25, -40) mm, rotated rx -180 ry 0 rz 0.01 deg; joints [33.279, -40.27, 94.858, -141.394, 61.608, 160.183]
  MoveC 3685 to (-293.65, 181.36, -40) mm, rotated rx -180 ry 0 rz 0.01 deg; joints [33.24, -40.182, 94.671, -141.402, 61.517, 160.133] to (-294.76, 179.52, -40) mm, rotated rx 180 ry 0 rz 0.01 deg; joints [33.163, -40.184, 94.679, -141.486, 61.493, 160.177]
  MoveL 3686 to (-294.76, 153.8, -40) mm, rotated rx 180 ry 0 rz 0.01 deg; joints [32.382, -40.822, 96.075, -142.567, 61.814, 161.11]
  MoveC 3687 to (-293.66, 149.33, -40) mm, rotated rx -180 ry 0 rz 0.01 deg; joints [32.266, -40.974, 96.405, -142.748, 61.916, 161.291] to (-290.62, 145.88, -40) mm, rotated rx 180 ry 0 rz 0.01 deg; joints [32.219, -41.177, 96.843, -142.874, 62.087, 161.476]
  MoveC 3688 to (-286.38, 142.89, -40) mm, rotated rx 180 ry 0 rz 0.01 deg; joints [32.209, -41.415, 97.354, -142.971, 62.302, 161.667] to (-282.16, 139.88, -40) mm, rotated rx 180 ry 0 rz 0.01 deg; joints [32.198, -41.652, 97.863, -143.069, 62.515, 161.858]
  MoveC 3689 to (-278.04, 136.73, -40) mm, rotated rx -180 ry 0 rz 0.01 deg; joints [32.181, -41.887, 98.369, -143.171, 62.726, 162.049] to (-274.1, 133.35, -40) mm, rotated rx 180 ry 0 rz 0.01 deg; joints [32.153, -42.118, 98.868, -143.284, 62.932, 162.244]
  MoveC 3690 to (-268.93, 128.31, -40) mm, rotated rx -180 ry 0 rz 0.01 deg; joints [32.097, -42.434, 99.552, -143.454, 63.208, 162.517] to (-264.11, 122.94, -40) mm, rotated rx 180 ry 0 rz 0.01 deg; joints [32.022, -42.742, 100.22, -143.64, 63.474, 162.792]
  MoveC 3691 to (-259.56, 117.34, -40) mm, rotated rx 180 ry 0 rz 0.01 deg; joints [31.935, -43.043, 100.873, -143.836, 63.73, 163.067] to (-255.16, 111.62, -40) mm, rotated rx -180 ry 0 rz 0.01 deg; joints [31.84, -43.339, 101.516, -144.037, 63.982, 163.34]
  MoveC 3692 to (-251.29, 106.11, -40) mm, rotated rx 180 ry 0 rz 0.01 deg; joints [31.741, -43.608, 102.103, -144.233, 64.209, 163.595] to (-247.75, 100.37, -40) mm, rotated rx -180 ry 0 rz 0.01 deg; joints [31.626, -43.868, 102.671, -144.44, 64.424, 163.848]
  MoveC 3693 to (-245.2, 95.81, -40) mm, rotated rx 180 ry 0 rz 0.01 deg; joints [31.529, -44.063, 103.098, -144.607, 64.585, 164.042] to (-242.77, 91.19, -40) mm, rotated rx 180 ry 0 rz 0.01 deg; joints [31.428, -44.254, 103.518, -144.777, 64.741, 164.235]
  MoveC 3694 to (-240.34, 86.56, -40) mm, rotated rx -180 ry 0 rz 0.01 deg; joints [31.325, -44.444, 103.935, -144.947, 64.897, 164.427] to (-237.8, 82.01, -40) mm, rotated rx -180 ry 0 rz 0.01 deg; joints [31.227, -44.636, 104.357, -145.112, 65.057, 164.618]
  MoveC 3695 to (-234.69, 78.9, -40) mm, rotated rx -180 ry 0 rz 0.01 deg; joints [31.186, -44.816, 104.752, -145.212, 65.221, 164.771] to (-230.45, 77.76, -40) mm, rotated rx 180 ry 0 rz 0.01 deg; joints [31.234, -44.996, 105.142, -145.217, 65.407, 164.882]
  MoveL 3696 to (-163.09, 77.76, -40) mm, rotated rx 180 ry 0 rz 0.01 deg; joints [32.635, -47.377, 110.308, -144.439, 68.068, 166.033]
  MoveC 3697 to (-158.84, 78.9, -40) mm, rotated rx -180 ry 0 rz 0.01 deg; joints [32.766, -47.499, 110.57, -144.336, 68.217, 166.069] to (-155.73, 82.01, -40) mm, rotated rx -180 ry 0 rz 0.01 deg; joints [32.939, -47.539, 110.652, -144.167, 68.297, 166.027]
  MoveC 3698 to (-153.11, 86.67, -40) mm, rotated rx -180 ry 0 rz 0.01 deg; joints [33.153, -47.529, 110.622, -143.939, 68.337, 165.93] to (-150.62, 91.39, -40) mm, rotated rx 180 ry 0 rz 0.01 deg; joints [33.367, -47.513, 110.578, -143.711, 68.371, 165.828]
  MoveC 3699 to (-148.12, 96.11, -40) mm, rotated rx 180 ry 0 rz 0.01 deg; joints [33.581, -47.497, 110.532, -143.483, 68.405, 165.725] to (-145.51, 100.77, -40) mm, rotated rx 180 ry 0 rz 0.01 deg; joints [33.795, -47.484, 110.496, -143.256, 68.444, 165.626]
  MoveC 3700 to (-136.92, 113.8, -40) mm, rotated rx -180 ry 0 rz 0.01 deg; joints [34.422, -47.489, 110.48, -142.603, 68.6, 165.369] to (-126.85, 125.71, -40) mm, rotated rx 180 ry 0 rz 0.01 deg; joints [35.046, -47.56, 110.613, -141.974, 68.821, 165.169]
  MoveC 3701 to (-115.49, 136.4, -40) mm, rotated rx -180 ry 0 rz 0.01 deg; joints [35.662, -47.694, 110.886, -141.374, 69.103, 165.027] to (-103.02, 145.78, -40) mm, rotated rx 180 ry 0 rz 0.01 deg; joints [36.264, -47.888, 111.29, -140.806, 69.437, 164.944]
  MoveC 3702 to (-99.89, 149.25, -40) mm, rotated rx -180 ry 0 rz 0.01 deg; joints [36.452, -47.91, 111.332, -140.619, 69.505, 164.887] to (-98.75, 153.78, -40) mm, rotated rx -180 ry 0 rz 0.01 deg; joints [36.626, -47.842, 111.175, -140.419, 69.486, 164.763]
  MoveL 3703 to (-98.76, 179.51, -40) mm, rotated rx 180 ry 0 rz 0.01 deg; joints [37.452, -47.236, 109.805, -139.39, 69.144, 163.93]
  MoveC 3704 to (-99.86, 181.37, -40) mm, rotated rx 180 ry 0 rz 0.01 deg; joints [37.484, -47.155, 109.626, -139.333, 69.079, 163.849] to (-102.02, 181.28, -40) mm, rotated rx -180 ry 0 rz 0.01 deg; joints [37.428, -47.087, 109.478, -139.369, 69.002, 163.814]
  MoveC 3705 to (-110.21, 176.26, -40) mm, rotated rx 180 ry 0 rz 0.01 deg; joints [37.072, -46.94, 109.167, -139.692, 68.77, 163.836] to (-118.66, 171.69, -40) mm, rotated rx 180 ry 0 rz 0.01 deg; joints [36.725, -46.771, 108.808, -139.999, 68.52, 163.837]
  MoveC 3706 to (-127.39, 167.68, -40) mm, rotated rx 180 ry 0 rz 0.01 deg; joints [36.392, -46.576, 108.392, -140.285, 68.25, 163.814] to (-136.41, 164.35, -40) mm, rotated rx -180 ry 0 rz 0.01 deg; joints [36.076, -46.353, 107.914, -140.544, 67.958, 163.764]
  MoveC 3707 to (-155.66, 159.67, -40) mm, rotated rx -180 ry 0 rz 0.01 deg; joints [35.486, -45.809, 106.746, -140.99, 67.294, 163.574] to (-175.39, 157.98, -40) mm, rotated rx -180 ry 0 rz 0.01 deg; joints [34.99, -45.166, 105.36, -141.304, 66.563, 163.274]
  MoveL 3708 to (-214.9, 157.8, -40) mm, rotated rx 180 ry 0 rz 0.01 deg; joints [34.127, -43.761, 102.338, -141.749, 65.024, 162.548]
  MoveC 3709 to (-237.75, 159.72, -40) mm, rotated rx 180 ry 0 rz 0.01 deg; joints [33.708, -42.872, 100.433, -141.888, 64.087, 162.045] to (-259.96, 165.43, -40) mm, rotated rx 180 ry 0 rz 0.01 deg; joints [33.429, -41.895, 98.336, -141.838, 63.114, 161.407]
  MoveC 3710 to (-262.96, 167.63, -40) mm, rotated rx 180 ry 0 rz 0.01 deg; joints [33.436, -41.726, 97.973, -141.77, 62.963, 161.269] to (-264.23, 171.13, -40) mm, rotated rx -180 ry 0 rz 0.01 deg; joints [33.517, -41.591, 97.68, -141.634, 62.867, 161.119]
  MoveC 3711 to (-265.43, 174.63, -40) mm, rotated rx 180 ry 0 rz 0.01 deg; joints [33.6, -41.458, 97.392, -141.498, 62.774, 160.97] to (-268.29, 176.97, -40) mm, rotated rx 180 ry 0 rz 0.01 deg; joints [33.613, -41.289, 97.028, -141.421, 62.627, 160.827]
  MoveC 3712 to (-272.04, 178.65, -40) mm, rotated rx 180 ry 0 rz 0.01 deg; joints [33.589, -41.102, 96.627, -141.378, 62.451, 160.689] to (-275.74, 180.44, -40) mm, rotated rx 180 ry 0 rz 0.01 deg; joints [33.569, -40.913, 96.222, -141.328, 62.275, 160.547]
  MoveC 3713 to (-282.03, 183.93, -40) mm, rotated rx 180 ry 0 rz 0.01 deg; joints [33.548, -40.578, 95.506, -141.224, 61.971, 160.287] to (-288, 187.94, -40) mm, rotated rx -180 ry 0 rz 0.01 deg; joints [33.55, -40.24, 94.783, -141.093, 61.671, 160.012]
  MoveC 3714 to (-293.74, 192.26, -40) mm, rotated rx 180 ry 0 rz 0.01 deg; joints [33.565, -39.9, 94.057, -140.945, 61.376, 159.728] to (-299.4, 196.68, -40) mm, rotated rx 180 ry 0 rz 0.01 deg; joints [33.585, -39.559, 93.326, -140.789, 61.082, 159.438]
  MoveC 3715 to (-301.46, 196.92, -40) mm, rotated rx 180 ry 0 rz 0.01 deg; joints [33.551, -39.469, 93.137, -140.79, 60.992, 159.383] to (-302.56, 195.16, -40) mm, rotated rx -180 ry 0 rz 0.01 deg; joints [33.477, -39.47, 93.142, -140.869, 60.967, 159.425]
  MoveL 3716 to (-302.56, 149.25, -40) mm, rotated rx -180 ry 0 rz 0.01 deg; joints [32.092, -40.622, 95.657, -142.806, 61.541, 161.11]
  MoveC 3717 to (-301.47, 144.96, -40) mm, rotated rx -180 ry 0 rz 0.01 deg; joints [31.981, -40.769, 95.977, -142.98, 61.641, 161.286] to (-298.45, 141.72, -40) mm, rotated rx 180 ry 0 rz 0.01 deg; joints [31.94, -40.967, 96.403, -143.098, 61.809, 161.463]
  MoveC 3718 to (-288.04, 134.33, -40) mm, rotated rx 180 ry 0 rz 0.01 deg; joints [31.912, -41.553, 97.662, -143.342, 62.338, 161.933] to (-278.37, 126, -40) mm, rotated rx 180 ry 0 rz 0.01 deg; joints [31.839, -42.124, 98.894, -143.623, 62.845, 162.412]
  MoveC 3719 to (-269.49, 116.83, -40) mm, rotated rx 180 ry 0 rz 0.01 deg; joints [31.724, -42.677, 100.09, -143.938, 63.327, 162.895] to (-261.41, 106.95, -40) mm, rotated rx 180 ry 0 rz 0.01 deg; joints [31.568, -43.207, 101.244, -144.285, 63.783, 163.378]
  MoveC 3720 to (-257.81, 101.81, -40) mm, rotated rx 180 ry 0 rz 0.01 deg; joints [31.474, -43.458, 101.79, -144.469, 63.995, 163.615] to (-254.51, 96.47, -40) mm, rotated rx 180 ry 0 rz 0.01 deg; joints [31.367, -43.7, 102.319, -144.664, 64.196, 163.851]
  MoveC 3721 to (-251.4, 90.94, -40) mm, rotated rx -180 ry 0 rz 0.01 deg; joints [31.249, -43.938, 102.84, -144.867, 64.391, 164.087] to (-248.41, 85.34, -40) mm, rotated rx 180 ry 0 rz 0.01 deg; joints [31.126, -44.171, 103.351, -145.074, 64.583, 164.322]
  MoveC 3722 to (-245.42, 79.74, -40) mm, rotated rx 180 ry 0 rz 0.01 deg; joints [31.001, -44.403, 103.86, -145.28, 64.774, 164.554] to (-242.31, 74.2, -40) mm, rotated rx 180 ry 0 rz 0.01 deg; joints [30.881, -44.636, 104.372, -145.482, 64.969, 164.785]
  MoveC 3723 to (-239.2, 71.09, -40) mm, rotated rx -180 ry 0 rz 0.01 deg; joints [30.84, -44.816, 104.766, -145.582, 65.134, 164.937] to (-234.96, 69.95, -40) mm, rotated rx 180 ry 0 rz 0.01 deg; joints [30.886, -44.996, 105.156, -145.588, 65.321, 165.047]
  MoveL 3724 to (-158.59, 69.95, -40) mm, rotated rx 180 ry 0 rz 0.01 deg; joints [32.468, -47.694, 111.014, -144.703, 68.342, 166.343]
  MoveC 3725 to (-154.34, 71.09, -40) mm, rotated rx 180 ry 0 rz 0.01 deg; joints [32.599, -47.814, 111.276, -144.6, 68.491, 166.379] to (-151.22, 74.2, -40) mm, rotated rx 180 ry 0 rz 0.01 deg; joints [32.773, -47.855, 111.359, -144.429, 68.57, 166.337]
  MoveL 3726 to (-138.75, 96.87, -40) mm, rotated rx -180 ry 0 rz 0.01 deg; joints [33.816, -47.795, 111.183, -143.322, 68.751, 165.86]
  MoveC 3727 to (-130.14, 109.76, -40) mm, rotated rx -180 ry 0 rz 0.01 deg; joints [34.442, -47.803, 111.175, -142.672, 68.907, 165.609] to (-119.94, 121.44, -40) mm, rotated rx 180 ry 0 rz 0.01 deg; joints [35.065, -47.884, 111.328, -142.047, 69.135, 165.42]
  MoveC 3728 to (-108.48, 131.86, -40) mm, rotated rx 180 ry 0 rz 0.01 deg; joints [35.678, -48.026, 111.62, -141.452, 69.421, 165.289] to (-96.05, 141.1, -40) mm, rotated rx -180 ry 0 rz 0.01 deg; joints [36.278, -48.22, 112.026, -140.886, 69.754, 165.21]
  MoveL 3729 to (-95.56, 141.41, -40) mm, rotated rx 180 ry 0 rz 0.01 deg; joints [36.3, -48.229, 112.045, -140.867, 69.768, 165.209]
  MoveL 3730 to (-95.07, 141.71, -40) mm, rotated rx 180 ry 0 rz 0.01 deg; joints [36.322, -48.238, 112.064, -140.847, 69.782, 165.208]
  MoveC 3731 to (-92.04, 144.99, -40) mm, rotated rx 180 ry 0 rz 0.01 deg; joints [36.502, -48.26, 112.107, -140.667, 69.848, 165.156] to (-90.95, 149.32, -40) mm, rotated rx 180 ry 0 rz 0.01 deg; joints [36.67, -48.196, 111.958, -140.475, 69.83, 165.038]
  MoveL 3732 to (-90.95, 195.18, -40) mm, rotated rx 180 ry 0 rz 0.01 deg; joints [38.137, -47.109, 109.5, -138.647, 69.217, 163.549]
  MoveC 3733 to (-92.06, 196.94, -40) mm, rotated rx 180 ry 0 rz 0.01 deg; joints [38.165, -47.03, 109.326, -138.594, 69.154, 163.471] to (-94.12, 196.72, -40) mm, rotated rx 180 ry 0 rz 0.01 deg; joints [38.107, -46.969, 109.193, -138.635, 69.083, 163.442]
  MoveC 3734 to (-101.31, 191.25, -40) mm, rotated rx -180 ry 0 rz 0.01 deg; joints [37.76, -46.869, 108.986, -138.962, 68.895, 163.497] to (-108.7, 186.07, -40) mm, rotated rx 180 ry 0 rz 0.01 deg; joints [37.418, -46.753, 108.744, -139.278, 68.695, 163.538]
  MoveC 3735 to (-116.4, 181.33, -40) mm, rotated rx 180 ry 0 rz 0.01 deg; joints [37.085, -46.614, 108.451, -139.58, 68.476, 163.559] to (-124.44, 177.22, -40) mm, rotated rx 180 ry 0 rz 0.01 deg; joints [36.764, -46.447, 108.094, -139.86, 68.233, 163.552]
  MoveC 3736 to (-134, 173.36, -40) mm, rotated rx 180 ry 0 rz 0.01 deg; joints [36.417, -46.219, 107.609, -140.149, 67.929, 163.51] to (-143.89, 170.45, -40) mm, rotated rx 180 ry 0 rz 0.01 deg; joints [36.096, -45.955, 107.042, -140.4, 67.598, 163.429]
  MoveC 3737 to (-153.96, 168.28, -40) mm, rotated rx 180 ry 0 rz 0.01 deg; joints [35.797, -45.664, 106.415, -140.62, 67.247, 163.32] to (-164.13, 166.61, -40) mm, rotated rx 180 ry 0 rz 0.01 deg; joints [35.514, -45.353, 105.748, -140.816, 66.883, 163.192]
  MoveC 3738 to (-171.35, 165.85, -40) mm, rotated rx -180 ry 0 rz 0.01 deg; joints [35.328, -45.12, 105.247, -140.935, 66.616, 163.085] to (-178.62, 165.6, -40) mm, rotated rx -180 ry 0 rz 0.01 deg; joints [35.159, -44.872, 104.713, -141.032, 66.341, 162.961]
  MoveL 3739 to (-214.9, 165.6, -40) mm, rotated rx 180 ry 0 rz 0.01 deg; joints [34.371, -43.574, 101.924, -141.428, 64.925, 162.282]
  MoveC 3740 to (-230.66, 166.57, -40) mm, rotated rx 180 ry 0 rz 0.01 deg; joints [34.068, -42.971, 100.631, -141.541, 64.285, 161.946] to (-246.18, 169.48, -40) mm, rotated rx -180 ry 0 rz 0.01 deg; joints [33.835, -42.319, 99.235, -141.559, 63.624, 161.54]
  MoveC 3741 to (-257.39, 172.78, -40) mm, rotated rx 180 ry 0 rz 0.01 deg; joints [33.707, -41.813, 98.149, -141.513, 63.127, 161.199] to (-268.29, 176.97, -40) mm, rotated rx 180 ry 0 rz 0.01 deg; joints [33.613, -41.289, 97.028, -141.421, 62.627, 160.827]
  MoveC 3742 to (-271.06, 179.34, -40) mm, rotated rx -180 ry 0 rz 0.01 deg; joints [33.629, -41.122, 96.67, -141.342, 62.483, 160.684] to (-272, 182.87, -40) mm, rotated rx -180 ry 0 rz 0.01 deg; joints [33.717, -40.998, 96.399, -141.201, 62.4, 160.537]
  MoveC 3743 to (-272.84, 186.39, -40) mm, rotated rx 180 ry 0 rz 0.01 deg; joints [33.807, -40.876, 96.134, -141.06, 62.321, 160.391] to (-275.4, 188.95, -40) mm, rotated rx -180 ry 0 rz 0.01 deg; joints [33.832, -40.711, 95.78, -140.971, 62.183, 160.244]
  MoveC 3744 to (-292.32, 200.36, -40) mm, rotated rx -180 ry 0 rz 0.01 deg; joints [33.834, -39.747, 93.72, -140.596, 61.334, 159.456] to (-307.13, 214.39, -40) mm, rotated rx 180 ry 0 rz 0.01 deg; joints [33.954, -38.777, 91.647, -140.078, 60.531, 158.587]
  MoveC 3745 to (-309.02, 214.86, -40) mm, rotated rx 180 ry 0 rz 0.01 deg; joints [33.931, -38.688, 91.457, -140.066, 60.445, 158.526] to (-310.12, 213.26, -40) mm, rotated rx -180 ry 0 rz 0.01 deg; joints [33.863, -38.685, 91.455, -140.139, 60.418, 158.562]
  MoveL 3746 to (-310.11, 144.71, -40) mm, rotated rx -180 ry 0 rz 0.01 deg; joints [31.809, -40.428, 95.255, -143.04, 61.276, 161.114]
  MoveC 3747 to (-309, 140.54, -40) mm, rotated rx 180 ry 0 rz 0.01 deg; joints [31.702, -40.574, 95.57, -143.21, 61.375, 161.287] to (-305.96, 137.47, -40) mm, rotated rx -180 ry 0 rz 0.01 deg; joints [31.665, -40.769, 95.99, -143.322, 61.543, 161.459]
  MoveC 3748 to (-295.03, 130.25, -40) mm, rotated rx 180 ry 0 rz 0.01 deg; joints [31.65, -41.374, 97.289, -143.559, 62.095, 161.935] to (-284.95, 121.88, -40) mm, rotated rx 180 ry 0 rz 0.01 deg; joints [31.582, -41.964, 98.56, -143.843, 62.621, 162.424]
  MoveC 3749 to (-275.77, 112.55, -40) mm, rotated rx 180 ry 0 rz 0.01 deg; joints [31.466, -42.533, 99.791, -144.166, 63.12, 162.919] to (-267.46, 102.43, -40) mm, rotated rx 180 ry 0 rz 0.01 deg; joints [31.305, -43.079, 100.976, -144.525, 63.589, 163.415]
  MoveC 3750 to (-264.11, 97.66, -40) mm, rotated rx -180 ry 0 rz 0.01 deg; joints [31.217, -43.312, 101.484, -144.696, 63.786, 163.635] to (-261.06, 92.7, -40) mm, rotated rx 180 ry 0 rz 0.01 deg; joints [31.117, -43.537, 101.975, -144.878, 63.973, 163.853]
  MoveL 3751 to (-246.67, 66.65, -40) mm, rotated rx -180 ry 0 rz 0.01 deg; joints [30.546, -44.633, 104.381, -145.839, 64.884, 164.946]
  MoveC 3752 to (-243.56, 63.54, -40) mm, rotated rx -180 ry 0 rz 0.01 deg; joints [30.504, -44.813, 104.775, -145.94, 65.049, 165.098] to (-239.32, 62.4, -40) mm, rotated rx 180 ry 0 rz 0.01 deg; joints [30.549, -44.993, 105.165, -145.946, 65.236, 165.207]
  MoveL 3753 to (-154.23, 62.4, -40) mm, rotated rx 180 ry 0 rz 0.01 deg; joints [32.304, -47.997, 111.693, -144.959, 68.607, 166.639]
  MoveC 3754 to (-149.98, 63.54, -40) mm, rotated rx 180 ry 0 rz 0.01 deg; joints [32.436, -48.117, 111.954, -144.854, 68.755, 166.675] to (-146.87, 66.65, -40) mm, rotated rx 180 ry 0 rz 0.01 deg; joints [32.61, -48.158, 112.038, -144.682, 68.835, 166.634]
  MoveL 3755 to (-132.21, 93.09, -40) mm, rotated rx -180 ry 0 rz 0.01 deg; joints [33.836, -48.094, 111.845, -143.385, 69.048, 166.084]
  MoveC 3756 to (-123.32, 106.3, -40) mm, rotated rx 180 ry 0 rz 0.01 deg; joints [34.483, -48.105, 111.841, -142.714, 69.208, 165.83] to (-112.7, 118.18, -40) mm, rotated rx 180 ry 0 rz 0.01 deg; joints [35.126, -48.193, 112.012, -142.072, 69.447, 165.643]
  MoveC 3757 to (-100.67, 128.6, -40) mm, rotated rx -180 ry 0 rz 0.01 deg; joints [35.756, -48.353, 112.341, -141.464, 69.752, 165.523] to (-87.49, 137.53, -40) mm, rotated rx -180 ry 0 rz 0.01 deg; joints [36.368, -48.576, 112.812, -140.894, 70.113, 165.467]
  MoveC 3758 to (-84.49, 140.59, -40) mm, rotated rx -180 ry 0 rz 0.01 deg; joints [36.541, -48.602, 112.864, -140.722, 70.18, 165.422] to (-83.4, 144.74, -40) mm, rotated rx -180 ry 0 rz 0.01 deg; joints [36.704, -48.543, 112.726, -140.538, 70.164, 165.311]
  MoveL 3759 to (-83.4, 213.26, -40) mm, rotated rx -180 ry 0 rz 0.01 deg; joints [38.887, -46.904, 109.024, -137.816, 69.247, 163.077]
